           "AC".CTL_AV_OFFS_TD := "AM_PAR_INTERPOL" (x:=#act_x, phase:= #act_phase, interpol:= #act_interpol,
                           x_par:="PAR_X_VALUES_7".PAR, y_par:="PAR_CTL_OFFS_AVR_TD".PAR);

           "AC".CTL_AV_OFFS_T1 := "AM_PAR_INTERPOL" (x:=#act_x, phase:= #act_phase, interpol:= #act_interpol,
                           x_par:="PAR_X_VALUES_7".PAR, y_par:="PAR_CTL_OFFS_AVR_T1".PAR);
       END_IF;
END_FUNCTION

FUNCTION "AM_PAR_FNC_CAM" : Void   // FC234, SCL
{ S7_Optimized_Access := 'FALSE' }
VERSION : 0.0
// --------------------------------------------------------------------------------
//     program     :    AM_PAR_FNC_CAM
//     description :    Calculate all camera setpoints from function tables.
//     name        :    D.Bruess
//     date        :    21.10.99
// 
//     revision    :    1.00
//     name        :    D.Bruess
//     date        :    21.10.99
//                     (c) CGS
//     --------------------------------------------------------------------------------
   VAR_INPUT
      act_x : Real;   // actual x value, x > 0
      act_phase : Int;   // process phase, 0 ... 9
      act_interpol : Bool;   // TRUE = with interpolation
   END_VAR
   VAR_TEMP
      YAct : Real;
   END_VAR
BEGIN


       //refresh camera parameters from recipe tables in one second cycle
       //----------------------------------------------------------------
       IF "SysTick1s" THEN   
           "AC".SET_SEN_THR    := "AM_PAR_INTERPOL" (x:=#act_x, phase:= #act_phase, interpol:= #act_interpol,
                           x_par:="PAR_X_VALUES_10".PAR, y_par:="PAR_CAM_THR".PAR);

           "AC".SET_SEN_WDH    := "AM_PAR_INTERPOL" (x:=#act_x, phase:= #act_phase, interpol:= #act_interpol,
                        x_par:="PAR_X_VALUES_10".PAR, y_par:="PAR_CAM_WIN_SIZE_H".PAR);

           "AC".SET_SEN_HGT    := "AM_PAR_INTERPOL" (x:=#act_x, phase:= #act_phase, interpol:= #act_interpol,
                        x_par:="PAR_X_VALUES_10".PAR, y_par:="PAR_CAM_WIN_SIZE_V".PAR);

           "AC".SET_SEN_CTR_X  := "AM_PAR_INTERPOL" (x:=#act_x, phase:= #act_phase, interpol:= #act_interpol,
                        x_par:="PAR_X_VALUES_10".PAR, y_par:="PAR_CAM_WIN_POS_H".PAR);

           "AC".SET_SEN_CTR_Y  := "AM_PAR_INTERPOL" (x:=#act_x, phase:= #act_phase, interpol:= #act_interpol,
                        x_par:="PAR_X_VALUES_10".PAR, y_par:="PAR_CAM_WIN_POS_V".PAR);

           "AC".SET_SEN_OUT_RAD  := "AM_PAR_INTERPOL" (x:=#act_x, phase:= #act_phase, interpol:= #act_interpol,
                                                   x_par:="PAR_X_VALUES_10".PAR, y_par:="PAR_CAM_SET_OUT_RAD".PAR);

           "AC".SET_SEN_IN_RAD   := "AM_PAR_INTERPOL" (x:=#act_x, phase:= #act_phase, interpol:= #act_interpol,
                                                   x_par:="PAR_X_VALUES_10".PAR, y_par:="PAR_CAM_SET_IN_RAD".PAR);

           "AC".SET_SEN_SEQ_STR_AGL  := "AM_PAR_INTERPOL" (x:=#act_x, phase:= #act_phase, interpol:= #act_interpol,
                                                       x_par:="PAR_X_VALUES_10".PAR, y_par:="PAR_CAM_SET_SEQ_STR_AGL".PAR);

           "AC".SET_SEN_SEQ_STP_AGL  := "AM_PAR_INTERPOL" (x:=#act_x, phase:= #act_phase, interpol:= #act_interpol,
                                                       x_par:="PAR_X_VALUES_10".PAR, y_par:="PAR_CAM_SET_SEQ_STP_AGL".PAR);


           IF ((#act_phase ="APC".NECK) OR (#act_phase ="APC".SHOULDER) OR (#act_phase ="APC".BODY)) THEN

               "AC".XT_MENISCUS := "AM_PAR_INTERPOL"(x:=#act_x, phase:= #act_phase, interpol:= #act_interpol,
                                                   x_par:="PAR_X_VALUES_10".PAR, y_par:="PAR_XT_MEN".PAR);

           ELSE
               "AC".XT_MENISCUS := 0.0;
           END_IF;

           //stereo camera
           //-------------
           "AC".SET_ROI_CTR_X_SCAM   := "AM_PAR_INTERPOL" (x:=#act_x, phase:= #act_phase, interpol:= #act_interpol,
                        x_par:="PAR_X_VALUES_10".PAR, y_par:="PAR_SCAM_CTR_X_POS".PAR);

           "AC".SET_ROI_CTR_Y_SCAM   := "AM_PAR_INTERPOL" (x:=#act_x, phase:= #act_phase, interpol:= #act_interpol,
                        x_par:="PAR_X_VALUES_10".PAR, y_par:="PAR_SCAM_CTR_Y_POS".PAR);

           "AC".SET_CAM_2_THR    := "AM_PAR_INTERPOL" (x:=#act_x, phase:= #act_phase, interpol:= #act_interpol,
                           x_par:="PAR_X_VALUES_10".PAR, y_par:="PAR_CAM_2_THR".PAR);

       END_IF;
END_FUNCTION

FUNCTION "AM_PAR_FNC_AV_CR_ROT_CTL" : Void   // FC235, SCL
{ S7_Optimized_Access := 'FALSE' }
VERSION : 0.0
// --------------------------------------------------------------------------------
//     program     :    AM_PAR_FNC_AV_CR_ROT_CTL
//     description :    Calculate all pid parameter for average crucible rotation 
//                      control loop from function tables.
//     name        :    G. Eibelsh鋟ser
//     date        :    11.01.2001
// 
//     revision    :    
//     name        :    
//     date        :    
//                     (c) CGS
//     --------------------------------------------------------------------------------
   VAR_INPUT
      act_x : Real;   // actual x value, x > 0
      act_phase : Int;   // process phase, 0 ... 9
      act_interpol : Bool;   // TRUE = with interpolation
   END_VAR
   VAR_TEMP
      YAct : Real;
   END_VAR
BEGIN


      "AC".CTL_AV_CRUC_ROT_GN := "AM_PAR_INTERPOL" (x:=#act_x, phase:= #act_phase, interpol:= #act_interpol,
                            x_par:="PAR_X_VALUES_8".PAR, y_par:="PAR_CTRL_AV_CRUC_ROT_GN".PAR);

      "AC".CTL_AV_CRUC_ROT_TI := "AM_PAR_INTERPOL" (x:=#act_x, phase:= #act_phase, interpol:= #act_interpol,
                            x_par:="PAR_X_VALUES_8".PAR, y_par:="PAR_CTRL_AV_CRUC_ROT_TI".PAR);

      "AC".CTL_AV_CRUC_ROT_TD := "AM_PAR_INTERPOL" (x:=#act_x, phase:= #act_phase, interpol:= #act_interpol,
                            x_par:="PAR_X_VALUES_8".PAR, y_par:="PAR_CTRL_AV_CRUC_ROT_TD".PAR);

      "AC".CTL_AV_CRUC_ROT_T1 := "AM_PAR_INTERPOL" (x:=#act_x, phase:= #act_phase, interpol:= #act_interpol,
                            x_par:="PAR_X_VALUES_8".PAR, y_par:="PAR_CTRL_AV_CRUC_ROT_T1".PAR);
END_FUNCTION

FUNCTION "AM_PAR_FNC_PD" : Void   // FC240, SCL
{ S7_Optimized_Access := 'FALSE' }
VERSION : 0.0
// --------------------------------------------------------------------------------
//     program     :    AM_PAR_FNC_PD
//     description :    Calculate all from function tables for PUMP DOWN process.
//     name        :    D.Bruess
//     date        :    21.10.99
// 
//     revision    :    1.00
//     name        :    D.Bruess
//     date        :    21.10.99
//                     (c) CGS
//     --------------------------------------------------------------------------------
   VAR_INPUT
      act_x_value : Real;   // actual x value, x > 0
   END_VAR
   VAR_TEMP
      YAct : Real;
      act_phase_number : Int;
   END_VAR
BEGIN


     #act_phase_number := "APC".PUMP_DOWN;

     // main page
     // ---------
     "AM_SET_V2" (act_phase := #act_phase_number);
     "AC".XT_MENISCUS := 0.0;

     // page 1
     // ------

     // page 2
     // ------

     // page 3
     // ------

     // page 4
     // ------

     // page 5
     // ------

     // page 6
     // ------

     // page 7
     // ------

     // page 8
     // ------

     // page 9
     // ------

     // page 10
     // ------
END_FUNCTION

FUNCTION "AM_PAR_FNC_ME" : Void   // FC241, SCL
{ S7_Optimized_Access := 'FALSE' }
VERSION : 0.0
// --------------------------------------------------------------------------------
//     program     :    AM_PAR_FNC_ME
//     description :    Calculate all from function tables for MELTING process.
//     name        :    D.Bruess
//     date        :    21.10.99
// 
//     revision    :    1.00
//     name        :    D.Bruess
//     date        :    21.10.99
//                     (c) CGS
//     --------------------------------------------------------------------------------
   VAR_INPUT
      act_x_value : Real;   // actual x value, x > 0
   END_VAR
   VAR_TEMP
      YAct : Real;
      act_phase_number : Int;
   END_VAR
BEGIN


     #act_phase_number := "APC".MELTING;

     // main page
     // ---------
     "AM_SET_V2" (act_phase := #act_phase_number);

     // page 1
     // ------
   (*YAct := AM_PAR_INTERPOL 
               (x:=act_x_value, phase:= act_phase_number, interpol:= FALSE,
                      x_par:=PAR_X_VALUES_1.PAR, y_par:=PAR_TIME.PAR);   *)

     "AV".SET_CR_POS := "AM_PAR_INTERPOL" 
               (x:=#act_x_value, phase:= #act_phase_number, interpol:= FALSE,
                      x_par:="PAR_X_VALUES_1".PAR, y_par:="PAR_CR_POS".PAR);

     "AV".SET_CR_SPD := "AM_PAR_INTERPOL" 
               (x:=#act_x_value, phase:= #act_phase_number, interpol:= FALSE,
                      x_par:="PAR_X_VALUES_1".PAR, y_par:="PAR_CR_SPD".PAR);

     "AC".SET_HTR_1_PWR := "AM_PAR_INTERPOL" 
               (x:=#act_x_value, phase:= #act_phase_number, interpol:= FALSE,
                      x_par:="PAR_X_VALUES_1".PAR, y_par:="PAR_HTR_1_PWR".PAR);

     "AC".SET_HTR_2_PWR := "AM_PAR_INTERPOL" 
               (x:=#act_x_value, phase:= #act_phase_number, interpol:= FALSE,
                      x_par:="PAR_X_VALUES_1".PAR, y_par:="PAR_HTR_2_PWR".PAR);

     "AC".SET_MOB_FDR_VIB_FRQ := "AM_PAR_INTERPOL" 
               (x:=#act_x_value, phase:= #act_phase_number, interpol:= FALSE,
                      x_par:="PAR_X_VALUES_1".PAR, y_par:="PAR_FDR_VIB_FRQ".PAR);





     // page 2
     // ------  

     // page 3
     // ------  
     "AM_PAR_FNC_ROT"
               (act_x:=#act_x_value, act_phase:=#act_phase_number, act_interpol:=FALSE);

     // page 4
     // ------
     "AM_PAR_FNC_GAS"
               (act_x:=#act_x_value, act_phase:=#act_phase_number, act_interpol:=FALSE);

     // page 5
     // ------
     "AM_PAR_FNC_MAG"
               (act_x:=#act_x_value, act_phase:=#act_phase_number, act_interpol:=FALSE);

     // page 6
     // ------

     // page 7
     // ------

     // page 8
     // ------

     // page 9
     // ------

     // page 10
     // ------
     "AM_PAR_FNC_CAM"
               (act_x:=#act_x_value, act_phase:=#act_phase_number, act_interpol:=FALSE);
END_FUNCTION

FUNCTION "AM_PAR_FNC_DI" : Void   // FC242, SCL
{ S7_Optimized_Access := 'FALSE' }
VERSION : 0.0
// --------------------------------------------------------------------------------
//     program     :    AM_PAR_FNC_DI
//     description :    Calculate all from function tables for DIPPING process.
//     name        :    D.Bruess
//     date        :    22.10.99
// 
//     revision    :    1.00
//     name        :    D.Bruess
//     date        :    22.10.99
//                     (c) CGS
//     --------------------------------------------------------------------------------
   VAR_INPUT
      act_x_value : Real;   // actual x value, x > 0
   END_VAR
   VAR_TEMP
      YAct : Real;
      act_phase_number : Int;
   END_VAR
BEGIN


     #act_phase_number := "APC".DIPPING;

     // main page
     // ---------
     "AM_SET_V2" (act_phase := #act_phase_number);

     // page 1
     // ------
   (*YAct := AM_PAR_INTERPOL (x:=act_x_value, phase:= act_phase_number, interpol:= FALSE,
                      x_par:=PAR_X_VALUES_1.PAR, y_par:=PAR_TIME.PAR);   *)

     // page 2
     // ------                 

     // page 3
     // ------  
     "AM_PAR_FNC_ROT"
               (act_x:=#act_x_value, act_phase:=#act_phase_number, act_interpol:=FALSE);

     // page 4
     // ------
     "AM_PAR_FNC_GAS" 
               (act_x:=#act_x_value, act_phase:=#act_phase_number, act_interpol:=FALSE);

     // page 5
     // ------
     "AM_PAR_FNC_MAG"
               (act_x:=#act_x_value, act_phase:=#act_phase_number, act_interpol:=FALSE);

     // page 6
     // ------

     // page 7
     // ------
     "AC".CTL_MLT_TMP_1_GN := "AM_PAR_INTERPOL" 
               (x:=#act_x_value, phase:= #act_phase_number, interpol:= FALSE,
                      x_par:="PAR_X_VALUES_7".PAR, y_par:="PAR_CTRL_MLT_TMP_1_GN".PAR);

     "AC".CTL_MLT_TMP_1_TI := "AM_PAR_INTERPOL" 
               (x:=#act_x_value, phase:= #act_phase_number, interpol:= FALSE,
                      x_par:="PAR_X_VALUES_7".PAR, y_par:="PAR_CTRL_MLT_TMP_1_TI".PAR);

     "AC".CTL_MLT_TMP_1_TD := "AM_PAR_INTERPOL"
               (x:=#act_x_value, phase:= #act_phase_number, interpol:= FALSE,
                      x_par:="PAR_X_VALUES_7".PAR, y_par:="PAR_CTRL_MLT_TMP_1_TD".PAR);

     "AC".CTL_MLT_TMP_1_T1 := "AM_PAR_INTERPOL"
               (x:=#act_x_value, phase:= #act_phase_number, interpol:= FALSE,
                      x_par:="PAR_X_VALUES_7".PAR, y_par:="PAR_CTRL_MLT_TMP_1_T1".PAR);

     // page 8
     // ------                 

     // page 9
     // ------
     "AC".PWR_COEFF_2 := "AM_PAR_INTERPOL" 
               (x:=#act_x_value, phase:= #act_phase_number, interpol:= FALSE,
                      x_par:="PAR_X_VALUES_9".PAR, y_par:="PAR_PWR_COEFF_2".PAR);

     // page 10
     // ------
     "AM_PAR_FNC_CAM" 
               (act_x:=#act_x_value, act_phase:=#act_phase_number, act_interpol:=FALSE);
END_FUNCTION

FUNCTION "AM_PAR_FNC_NE" : Void   // FC243, SCL
{ S7_Optimized_Access := 'FALSE' }
VERSION : 0.0
// --------------------------------------------------------------------------------
//     program     :    AM_PAR_FNC_NE
//     description :    Calculate all from function tables for NECK process.
//     name        :    D.Bruess
//     date        :    22.10.99
// 
//     revision    :    1.00
//     name        :    D.Bruess
//     date        :    22.10.99
//                     (c) CGS
//     --------------------------------------------------------------------------------
   VAR_INPUT
      act_x_value : Real;   // actual x value, x > 0
   END_VAR
   VAR_TEMP
      YAct : Real;
      act_phase_number : Int;
   END_VAR
BEGIN


     #act_phase_number := "APC".NECK;

     // main page
     // ---------
     "AM_SET_V2" (act_phase := #act_phase_number);

     // page 1
     // ------
     "AC".SET_AVG_SPD := "AM_PAR_INTERPOL" 
               (x:=#act_x_value, phase:= #act_phase_number, interpol:= TRUE,
                      x_par:="PAR_X_VALUES_1".PAR, y_par:="PAR_AV_SPD".PAR);

     "AC".SET_XT_SPD_DEV_1 := "AM_PAR_INTERPOL" 
               (x:=#act_x_value, phase:= #act_phase_number, interpol:= TRUE,
                      x_par:="PAR_X_VALUES_1".PAR, y_par:="PAR_AV_SPD_DEV_1".PAR);

     "AC".SET_XT_SPD_DEV_2 := "AM_PAR_INTERPOL" 
               (x:=#act_x_value, phase:= #act_phase_number, interpol:= TRUE,
                      x_par:="PAR_X_VALUES_1".PAR, y_par:="PAR_AV_SPD_DEV_2".PAR);

     "AV".SET_HTR_1_TMP_INC := "AM_PAR_INTERPOL" 
               (x:=#act_x_value, phase:= #act_phase_number, interpol:= TRUE,
                      x_par:="PAR_X_VALUES_1".PAR, y_par:="PAR_HTR_1_TMP".PAR);

     "AV".SET_HTR_2_PWR_INC := "AM_PAR_INTERPOL" 
               (x:=#act_x_value, phase:= #act_phase_number, interpol:= TRUE,
                      x_par:="PAR_X_VALUES_1".PAR, y_par:="PAR_HTR_2_PWR".PAR);

     // page 2
     // ------
     "AV".SET_XT_DIA := "AM_PAR_INTERPOL" 
               (x:=#act_x_value, phase:= #act_phase_number, interpol:= TRUE,
                      x_par:="PAR_X_VALUES_2".PAR, y_par:="PAR_XT_DIA".PAR);

     // page 3
     // ------  
     "AM_PAR_FNC_ROT"
               (act_x:=#act_x_value, act_phase:=#act_phase_number, act_interpol:=TRUE);

     // page 4
     // ------
     "AM_PAR_FNC_GAS" 
               (act_x:=#act_x_value, act_phase:=#act_phase_number, act_interpol:=TRUE);

     // page 5
     // ------
     "AM_PAR_FNC_MAG"
               (act_x:=#act_x_value, act_phase:=#act_phase_number, act_interpol:=TRUE);

     // page 6
     // ------

     // page 7
     // ------
     "AM_PAR_FNC_CTL" 
               (act_x:=#act_x_value, act_phase:=#act_phase_number, act_interpol:=TRUE);

     // page 8
     // ------          

     // page 9
     // ------
     "AC".PWR_COEFF_2 := "AM_PAR_INTERPOL" 
               (x:=#act_x_value, phase:= #act_phase_number, interpol:= TRUE,
                      x_par:="PAR_X_VALUES_9".PAR, y_par:="PAR_PWR_COEFF_2".PAR);

     // page 10
     // ------
     "AM_PAR_FNC_CAM" 
               (act_x:=#act_x_value, act_phase:=#act_phase_number, act_interpol:= TRUE);
END_FUNCTION

FUNCTION "AM_PAR_FNC_SH" : Void   // FC244, SCL
{ S7_Optimized_Access := 'FALSE' }
VERSION : 0.0
// --------------------------------------------------------------------------------
//     program     :    AM_PAR_FNC_SH
//     description :    Calculate all from function tables for SHOULDER process.
//     name        :    D.Bruess
//     date        :    22.10.99
// 
//     revision    :    1.00
//     name        :    D.Bruess
//     date        :    22.10.99
//                     (c) CGS
//     --------------------------------------------------------------------------------
   VAR_INPUT
      act_x_value : Real;   // actual x value, x > 0
   END_VAR
   VAR_TEMP
      YAct : Real;
      act_phase_number : Int;
   END_VAR
BEGIN


     #act_phase_number := "APC".SHOULDER;

     // main page
     // ---------
     "AM_SET_V2" (act_phase := #act_phase_number);

     // page 1
     // ------
     "AC".SET_GRW_RTE := "AM_PAR_INTERPOL" 
               (x:=#act_x_value, phase:= #act_phase_number, interpol:= TRUE,
                      x_par:="PAR_X_VALUES_1".PAR, y_par:="PAR_XT_GRO".PAR);


     IF "DV".TRANS_SH_BY_FLAG AND "CNF".CONF_SH_PAR_FNCT THEN   //transition to body? SH-Par as function of length? 
       "AC".SET_XT_SPD := "PAR_MAIN".SH_BODY_TRANS_SPD;        
     ELSE                                                  
       "AC".SET_XT_SPD := "AM_PAR_INTERPOL" 
                (x:=#act_x_value, phase:= #act_phase_number, interpol:= TRUE,
                       x_par:="PAR_X_VALUES_1".PAR, y_par:="PAR_XT_SPD".PAR);
     END_IF;                    

     "AC".SET_AVG_CRUC_ROT := "AM_PAR_INTERPOL" 
               (x:=#act_x_value, phase:= #act_phase_number, interpol:= TRUE,
                      x_par:="PAR_X_VALUES_1".PAR, y_par:="PAR_AV_CRUC_ROT".PAR);

     "AC".SET_CRUC_ROT_DEV_1 := "AM_PAR_INTERPOL" 
               (x:=#act_x_value, phase:= #act_phase_number, interpol:= TRUE,
                      x_par:="PAR_X_VALUES_1".PAR, y_par:="PAR_AV_CRUC_ROT_DEV_1".PAR);

     "AC".SET_CRUC_ROT_DEV_2 := "AM_PAR_INTERPOL" 
               (x:=#act_x_value, phase:= #act_phase_number, interpol:= TRUE,
                      x_par:="PAR_X_VALUES_1".PAR, y_par:="PAR_AV_CRUC_ROT_DEV_2".PAR);

     "AV".SET_HTR_1_TMP_INC := "AM_PAR_INTERPOL" 
               (x:=#act_x_value, phase:= #act_phase_number, interpol:= TRUE,
                      x_par:="PAR_X_VALUES_1".PAR, y_par:="PAR_HTR_1_TMP".PAR);

     "AV".SET_HTR_2_PWR_INC := "AM_PAR_INTERPOL" 
               (x:=#act_x_value, phase:= #act_phase_number, interpol:= TRUE,
                      x_par:="PAR_X_VALUES_1".PAR, y_par:="PAR_HTR_2_PWR".PAR);

     // page 2
     // ------  

     // page 3
     // ------  
     "AM_PAR_FNC_ROT"
               (act_x:=#act_x_value, act_phase:=#act_phase_number, act_interpol:=TRUE);

     // page 4
     // ------
     "AM_PAR_FNC_GAS" 
               (act_x:=#act_x_value, act_phase:=#act_phase_number, act_interpol:=TRUE);

     // page 5
     // ------
     "AM_PAR_FNC_MAG"
               (act_x:=#act_x_value, act_phase:=#act_phase_number, act_interpol:=TRUE);

     // page 6
     // ------
     "AC".SET_CR_SPD_COF := "AM_PAR_INTERPOL" 
               (x:=#act_x_value, phase:= #act_phase_number, interpol:= TRUE,
                      x_par:="PAR_X_VALUES_6".PAR, y_par:="PAR_CRSPD_COEFF".PAR);


     "AC".CTL_MLT_LVL_GN := "AM_PAR_INTERPOL" 
               (x:=#act_x_value, phase:= #act_phase_number, interpol:= TRUE,
                      x_par:="PAR_X_VALUES_6".PAR, y_par:="PAR_CTRL_MLT_LVL_GN".PAR);


     "AC".SET_MLT_LVL_INC := "AM_PAR_INTERPOL" 
               (x:=#act_x_value, phase:= #act_phase_number, interpol:= TRUE,
                      x_par:="PAR_X_VALUES_6".PAR, y_par:="PAR_MLT_LVL_INC".PAR);





     // page 7
     // ------
     "AC".CTL_GRO_GN := "AM_PAR_INTERPOL" 
               (x:=#act_x_value, phase:= #act_phase_number, interpol:= TRUE,
                      x_par:="PAR_X_VALUES_7".PAR, y_par:="PAR_CTRL_GRO_GN".PAR);

     "AC".CTL_GRO_TI := "AM_PAR_INTERPOL" 
               (x:=#act_x_value, phase:= #act_phase_number, interpol:= TRUE,
                      x_par:="PAR_X_VALUES_7".PAR, y_par:="PAR_CTRL_GRO_TI".PAR);

     "AC".CTL_GRO_TD := "AM_PAR_INTERPOL" 
               (x:=#act_x_value, phase:= #act_phase_number, interpol:= TRUE,
                      x_par:="PAR_X_VALUES_7".PAR, y_par:="PAR_CTRL_GRO_TD".PAR);

     "AC".CTL_GRO_T1 := "AM_PAR_INTERPOL" 
               (x:=#act_x_value, phase:= #act_phase_number, interpol:= TRUE,
                      x_par:="PAR_X_VALUES_7".PAR, y_par:="PAR_CTRL_GRO_T1".PAR);

     // page 8
     // ------
     "AM_PAR_FNC_AV_CR_ROT_CTL" 
               (act_x:=#act_x_value, act_phase:=#act_phase_number, act_interpol:=TRUE);

     // page 9
     // ------
     "AC".PWR_COEFF_2 := "AM_PAR_INTERPOL" 
               (x:=#act_x_value, phase:= #act_phase_number, interpol:= TRUE,
                      x_par:="PAR_X_VALUES_9".PAR, y_par:="PAR_PWR_COEFF_2".PAR);

     // page 10
     // -------
     "AM_PAR_FNC_CAM" 
               (act_x:=#act_x_value, act_phase:=#act_phase_number, act_interpol:= TRUE);
END_FUNCTION

FUNCTION "AM_PAR_FNC_BY" : Void   // FC245, SCL
{ S7_Optimized_Access := 'FALSE' }
VERSION : 0.0
// --------------------------------------------------------------------------------
//     program     :    AM_PAR_FNC_BY
//     description :    Calculate all from function tables for BODY process.
//     name        :    D.Bruess
//     date        :    22.10.99
// 
//     revision    :    1.00
//     name        :    D.Bruess
//     date        :    22.10.99
//                     (c) CGS
//     --------------------------------------------------------------------------------
   VAR_INPUT
      act_x_value : Real;   // actual x value, x > 0
   END_VAR
   VAR_TEMP
      YAct : Real;
      act_phase_number : Int;
   END_VAR
BEGIN


     #act_phase_number := "APC".BODY;

     // main page
     // ---------
     "AM_SET_V2" (act_phase := #act_phase_number);

     // page 1
     // ------
     "AC".SET_AVG_SPD := "AM_PAR_INTERPOL" 
               (x:=#act_x_value, phase:= #act_phase_number, interpol:= TRUE,
                      x_par:="PAR_X_VALUES_1".PAR, y_par:="PAR_AV_SPD".PAR);

     "AC".SET_XT_SPD_DEV_1 := "AM_PAR_INTERPOL" 
               (x:=#act_x_value, phase:= #act_phase_number, interpol:= TRUE,
                      x_par:="PAR_X_VALUES_1".PAR, y_par:="PAR_AV_SPD_DEV_1".PAR);

     "AC".SET_XT_SPD_DEV_2 := "AM_PAR_INTERPOL" 
               (x:=#act_x_value, phase:= #act_phase_number, interpol:= TRUE,
                      x_par:="PAR_X_VALUES_1".PAR, y_par:="PAR_AV_SPD_DEV_2".PAR);

     "AC".SET_AVG_CRUC_ROT := "AM_PAR_INTERPOL" 
               (x:=#act_x_value, phase:= #act_phase_number, interpol:= TRUE,
                      x_par:="PAR_X_VALUES_1".PAR, y_par:="PAR_AV_CRUC_ROT".PAR);

     "AC".SET_CRUC_ROT_DEV_1 := "AM_PAR_INTERPOL" 
               (x:=#act_x_value, phase:= #act_phase_number, interpol:= TRUE,
                      x_par:="PAR_X_VALUES_1".PAR, y_par:="PAR_AV_CRUC_ROT_DEV_1".PAR);

     "AC".SET_CRUC_ROT_DEV_2 := "AM_PAR_INTERPOL" 
               (x:=#act_x_value, phase:= #act_phase_number, interpol:= TRUE,
                      x_par:="PAR_X_VALUES_1".PAR, y_par:="PAR_AV_CRUC_ROT_DEV_2".PAR);

     "AV".SET_HTR_1_TMP_INC := "AM_PAR_INTERPOL" 
               (x:=#act_x_value, phase:= #act_phase_number, interpol:= TRUE,
                      x_par:="PAR_X_VALUES_1".PAR, y_par:="PAR_HTR_1_TMP".PAR);

     "AV".SET_HTR_2_PWR_INC := "AM_PAR_INTERPOL" 
               (x:=#act_x_value, phase:= #act_phase_number, interpol:= TRUE,
                      x_par:="PAR_X_VALUES_1".PAR, y_par:="PAR_HTR_2_PWR".PAR);

     // page 2
     // ------
     "AV".SET_XT_DIA := "AM_PAR_INTERPOL" 
               (x:=#act_x_value, phase:= #act_phase_number, interpol:= TRUE,
                      x_par:="PAR_X_VALUES_2".PAR, y_par:="PAR_XT_DIA".PAR);

     // page 3
     // ------  
     "AM_PAR_FNC_ROT"
               (act_x:=#act_x_value, act_phase:=#act_phase_number, act_interpol:=TRUE);

     // page 4
     // ------
     "AM_PAR_FNC_GAS" 
               (act_x:=#act_x_value, act_phase:=#act_phase_number, act_interpol:=TRUE);

     // page 5
     // ------
     "AM_PAR_FNC_MAG"
               (act_x:=#act_x_value, act_phase:=#act_phase_number, act_interpol:=TRUE);

     // page 6
     // ------
     "AC".SET_CR_SPD_COF := "AM_PAR_INTERPOL" 
               (x:=#act_x_value, phase:= #act_phase_number, interpol:= TRUE,
                      x_par:="PAR_X_VALUES_6".PAR, y_par:="PAR_CRSPD_COEFF".PAR);


     "AC".CTL_MLT_LVL_GN := "AM_PAR_INTERPOL" 
               (x:=#act_x_value, phase:= #act_phase_number, interpol:= TRUE,
                      x_par:="PAR_X_VALUES_6".PAR, y_par:="PAR_CTRL_MLT_LVL_GN".PAR);


     "AC".SET_MLT_LVL_INC := "AM_PAR_INTERPOL" 
               (x:=#act_x_value, phase:= #act_phase_number, interpol:= TRUE,
                      x_par:="PAR_X_VALUES_6".PAR, y_par:="PAR_MLT_LVL_INC".PAR);


     // page 7
     // ------
     "AM_PAR_FNC_CTL" 
               (act_x:=#act_x_value, act_phase:=#act_phase_number, act_interpol:=TRUE);

     // page 8
     // ------
     "AM_PAR_FNC_AV_CR_ROT_CTL" 
               (act_x:=#act_x_value, act_phase:=#act_phase_number, act_interpol:=TRUE);

     // page 9
     // ------
     "AC".PWR_COEFF_2 := "AM_PAR_INTERPOL" 
               (x:=#act_x_value, phase:= #act_phase_number, interpol:= TRUE,
                      x_par:="PAR_X_VALUES_9".PAR, y_par:="PAR_PWR_COEFF_2".PAR);

     // page 10
     // -------
     "AM_PAR_FNC_CAM" 
               (act_x:=#act_x_value, act_phase:=#act_phase_number, act_interpol:= TRUE);

       // page 11
       // -------
       "AC".CTL_DIA_TMP_GN :=    "AM_PAR_INTERPOL"(x           := #act_x_value, 
                                               phase       := #act_phase_number, 
                                               interpol    := TRUE,
                                               x_par       := "PAR_X_VALUES_11".PAR, 
                                               y_par       := "PAR_CTRL_DIA_TMP_GN".PAR);

       "AC".CTL_DIA_TMP_TI :=    "AM_PAR_INTERPOL"(x           := #act_x_value, 
                                               phase       := #act_phase_number, 
                                               interpol    := TRUE,
                                               x_par       := "PAR_X_VALUES_11".PAR, 
                                               y_par       := "PAR_CTRL_DIA_TMP_TI".PAR);

       "AC".CTL_DIA_TMP_TD :=    "AM_PAR_INTERPOL"(x           := #act_x_value, 
                                               phase       := #act_phase_number, 
                                               interpol    := TRUE,
                                               x_par       := "PAR_X_VALUES_11".PAR, 
                                               y_par       := "PAR_CTRL_DIA_TMP_TD".PAR);

       "AC".CTL_DIA_TMP_T1 :=    "AM_PAR_INTERPOL"(x           := #act_x_value, 
                                               phase       := #act_phase_number, 
                                               interpol    := TRUE,
                                               x_par       := "PAR_X_VALUES_11".PAR, 
                                               y_par       := "PAR_CTRL_DIA_TMP_T1".PAR);
END_FUNCTION

FUNCTION "AM_PAR_FNC_EC" : Void   // FC246, SCL
{ S7_Optimized_Access := 'FALSE' }
VERSION : 0.0
// --------------------------------------------------------------------------------
//     program     :    AM_PAR_FNC_EC
//     description :    Calculate all from function tables for ENDCONE process.
//     name        :    D.Bruess
//     date        :    22.10.99
// 
//     revision    :    1.00
//     name        :    D.Bruess
//     date        :    22.10.99
//                     (c) CGS
//     --------------------------------------------------------------------------------
   VAR_INPUT
      act_x_value : Real;   // actual x value, x > 0
   END_VAR
   VAR_TEMP
      YAct : Real;
      act_phase_number : Int;
   END_VAR
BEGIN


     #act_phase_number := "APC".ENDCONE;

     // main page
     // ---------
     "AM_SET_V2" (act_phase := #act_phase_number);

     // page 1
     // ------
     "AV".SET_XT_SPD := "AM_PAR_INTERPOL" 
               (x:=#act_x_value, phase:= #act_phase_number, interpol:= TRUE,
                      x_par:="PAR_X_VALUES_1".PAR, y_par:="PAR_XT_SPD".PAR);

     "AV".SET_CR_SPD := "AM_PAR_INTERPOL" 
               (x:=#act_x_value, phase:= #act_phase_number, interpol:= TRUE,
                      x_par:="PAR_X_VALUES_1".PAR, y_par:="PAR_CR_SPD".PAR);

     "AV".SET_HTR_1_TMP_INC := "AM_PAR_INTERPOL" 
               (x:=#act_x_value, phase:= #act_phase_number, interpol:= TRUE,
                      x_par:="PAR_X_VALUES_1".PAR, y_par:="PAR_HTR_1_TMP".PAR);

     "AV".SET_HTR_2_PWR_INC := "AM_PAR_INTERPOL" 
               (x:=#act_x_value, phase:= #act_phase_number, interpol:= TRUE,
                      x_par:="PAR_X_VALUES_1".PAR, y_par:="PAR_HTR_2_PWR".PAR);

     // page 2
     // ------  

     // page 3
     // ------
     "AM_PAR_FNC_ROT"
               (act_x:=#act_x_value, act_phase:=#act_phase_number, act_interpol:=TRUE);

     // page 4
     // ------
     "AM_PAR_FNC_GAS" 
               (act_x:=#act_x_value, act_phase:=#act_phase_number, act_interpol:=TRUE);

     // page 5
     // ------
     "AM_PAR_FNC_MAG"
               (act_x:=#act_x_value, act_phase:=#act_phase_number, act_interpol:=TRUE);

     // page 6
     // ------

     // page 7
     // ------

     // page 8
     // ------

     // page 9
     // ------
     "AC".PWR_COEFF_2 := "AM_PAR_INTERPOL" 
               (x:=#act_x_value, phase:= #act_phase_number, interpol:= TRUE,
                      x_par:="PAR_X_VALUES_9".PAR, y_par:="PAR_PWR_COEFF_2".PAR);

     // page 10
     // -------

     "AC".XT_MENISCUS := 0.0;
END_FUNCTION

FUNCTION "AM_PAR_FNC_SD" : Void   // FC247, SCL
{ S7_Optimized_Access := 'FALSE' }
VERSION : 0.0
// --------------------------------------------------------------------------------
//     program     :    AM_PAR_FNC_SD
//     description :    Calculate all from function tables for SHUT DOWN process.
//     name        :    D.Bruess
//     date        :    22.10.99
// 
//     revision    :    1.00
//     name        :    D.Bruess
//     date        :    22.10.99
//                     (c) CGS
//     --------------------------------------------------------------------------------
   VAR_INPUT
      act_x_value : Real;   // actual x value, x > 0
   END_VAR
   VAR_TEMP
      YAct : Real;
      act_phase_number : Int;
   END_VAR
BEGIN


     #act_phase_number := "APC".SHUT_DOWN;

     // main page
     // ---------
     "AM_SET_V2" (act_phase := #act_phase_number);

     // page 1
     // ------
   (*YAct := AM_PAR_INTERPOL 
               (x:=act_x_value, phase:= act_phase_number, interpol:= FALSE,
                      x_par:=PAR_X_VALUES_1.PAR, y_par:=PAR_TIME.PAR);   *)

     "AV".SET_XT_POS := "AM_PAR_INTERPOL" 
               (x:=#act_x_value, phase:= #act_phase_number, interpol:= FALSE,
                      x_par:="PAR_X_VALUES_1".PAR, y_par:="PAR_XT_POS".PAR);

     "AV".SET_XT_SPD := "AM_PAR_INTERPOL" 
               (x:=#act_x_value, phase:= #act_phase_number, interpol:= FALSE,
                      x_par:="PAR_X_VALUES_1".PAR, y_par:="PAR_XT_SPD".PAR);

     "AV".SET_CR_POS := "AM_PAR_INTERPOL" 
               (x:=#act_x_value, phase:= #act_phase_number, interpol:= FALSE,
                      x_par:="PAR_X_VALUES_1".PAR, y_par:="PAR_CR_POS".PAR);

     "AV".SET_CR_SPD := "AM_PAR_INTERPOL" 
               (x:=#act_x_value, phase:= #act_phase_number, interpol:= FALSE,
                      x_par:="PAR_X_VALUES_1".PAR, y_par:="PAR_CR_SPD".PAR);

     "AC".SET_HTR_1_PWR := "AM_PAR_INTERPOL" 
               (x:=#act_x_value, phase:= #act_phase_number, interpol:= FALSE,
                      x_par:="PAR_X_VALUES_1".PAR, y_par:="PAR_HTR_1_PWR".PAR);

     // page 2
     // ------  

     // page 3
     // ------
     "AM_PAR_FNC_ROT"
               (act_x:=#act_x_value, act_phase:=#act_phase_number, act_interpol:=FALSE);


     // page 4 (AV.xxx used for AM_PRS_CTRL() )
     // ------
     "AV".SET_GAS_1_FLW := "AM_PAR_INTERPOL"
               (x:=#act_x_value, phase:= #act_phase_number, interpol:= FALSE,
                      x_par:="PAR_X_VALUES_4".PAR, y_par:="PAR_GAS_1_FLW".PAR);

     "AV".SET_GAS_2_FLW := "AM_PAR_INTERPOL"
               (x:=#act_x_value, phase:= #act_phase_number, interpol:= FALSE,
                      x_par:="PAR_X_VALUES_4".PAR, y_par:="PAR_GAS_2_FLW".PAR);

     "AV".SET_PRS_FCH := "AM_PAR_INTERPOL"
               (x:=#act_x_value, phase:= #act_phase_number, interpol:= FALSE,
                      x_par:="PAR_X_VALUES_4".PAR, y_par:="PAR_PRS".PAR);

     // page 5
     // ------
     "AM_PAR_FNC_MAG"
               (act_x:=#act_x_value, act_phase:=#act_phase_number, act_interpol:=FALSE);

     // page 6
     // ------

     // page 7
     // ------

     // page 8
     // ------

     // page 9
     // ------
     "AC".PWR_COEFF_2 := "AM_PAR_INTERPOL" 
               (x:=#act_x_value, phase:= #act_phase_number, interpol:= FALSE,
                      x_par:="PAR_X_VALUES_9".PAR, y_par:="PAR_PWR_COEFF_2".PAR);

     // page 10
     // -------

     "AC".XT_MENISCUS := 0.0;
END_FUNCTION

FUNCTION "AM_PAR_FNC_RE" : Void   // FC248, SCL
{ S7_Optimized_Access := 'FALSE' }
VERSION : 0.0
// --------------------------------------------------------------------------------
//     program     :    AM_PAR_FNC_RE
//     description :    Calculate all from function tables for REMOVAL process.
//     name        :    G. Eibelsh鋟ser
//     date        :    31.07.2012
// 
//                     (c) PVA TePla AG
//     --------------------------------------------------------------------------------
   VAR_TEMP
      YAct : Real;
      act_phase_number : Int;
   END_VAR
BEGIN


     #act_phase_number := "APC".REMOVAL;

     // main page
     // ---------

     "AM_SET_V2" (act_phase := #act_phase_number);

     "AC".SET_GAS_1_FLW     := "PAR_MAIN".RC_GAS_1_FLW;
     "AC".SET_GAS_2_FLW     := "PAR_MAIN".RC_GAS_2_FLW;
     "AC".SET_CLF_PRS       := "PAR_MAIN".RC_PRS;

     "AV".SET_MAG_1_CUR     := "PAR_MAIN".RC_MAG_AV_CUR;
     "AV".SET_MAG_RATIO_CUR := "PAR_MAIN".RC_MAG_RATIO_CUR;
END_FUNCTION

FUNCTION "AM_PAR_INTERPOL" : Real   // FC254, SCL
{ S7_Optimized_Access := 'FALSE' }
VERSION : 0.0
// --------------------------------------------------------------------------------
//     program     :    AM_INTERPOLATION
//     description :    Calculate y value from x/y function table.
//     name        :    D.Bruess
//     date        :    18.10.99
// 
//     revision    :    process phase 1 ...10
//     name        :    D.Bruess
//     date        :    12.11.99
//                     (c) CGS
//     --------------------------------------------------------------------------------
   VAR_INPUT
      x : Real;   // actual x value, x > 0
      phase : Int;   // process phase, 1 ... 10
      interpol : Bool;   // TRUE = with interpolation
      x_par : Array[1..10, 1..21] of Real;   // array with x values
      y_par : Array[1..10, 1..21] of Real;   // array with y values
   END_VAR
   VAR_TEMP
      x1 : Real;
      x2 : Real;
      y1 : Real;
      y2 : Real;
      y : Real;
      i : Int;
      found : Int;
   END_VAR
BEGIN

     IF ((#phase > 10) OR (#phase < 1)) THEN       // invalid phase number ?
       #y := 0.0;
     ELSE;

       IF (#x < 0.0) THEN                        // invalid x value ?
         #y := #y_par[#phase,1];
       ELSE

         // search for interval
         #i := 1;
         #found := 0;

         WHILE #found = 0 DO

           #x1 := #x_par[#phase,#i];
           #x2 := #x_par[#phase,#i+1];
           #y1 := #y_par[#phase,#i];
           #y2 := #y_par[#phase,#i+1];

           IF (#x <= #x1) THEN                    // below x1 ?

             #y := #y1;  
             #found := 1;
           ELSE
             IF (#x < #x2) THEN                    // x1<x<x2 ?
               IF (#interpol = TRUE) THEN
                 #y := #y1 + ((#y2-#y1)/(#x2-#x1))*(#x-#x1);
               ELSE
                 #y := #y1;
               END_IF;
               #found := 1;

             ELSE                                 // x>=x2                           

               IF (#x2=0.0) THEN                   // last x[i] because next x=0 ?
                 #y := #y1;
                 #found := 1;
               ELSE
                 IF (#i = 20) THEN                 // last x[i] because i = 20 ?
                   #y := #y2;
                   #found := 1;

                 ELSE
                   #i := #i + 1;                    // next x[i]
                   #found := 0;

                 END_IF;

               END_IF;
              END_IF;
             END_IF;
           END_WHILE;
         END_IF;
       END_IF;


     #AM_PAR_INTERPOL := #y;
END_FUNCTION

FUNCTION "SM_RESTART_CALL" : Void   // FC256, SCL
{ S7_Optimized_Access := 'FALSE' }
VERSION : 0.0
// --------------------------------------------------------------------------------
//     program     :    SM_RESTART_CALL
//     description :    call functions for restart       
//     name        :    K. Kalkowski
//     date        :    04.11.98
// 
//     revision    :    
//     name        :
//     date        :    
//                     (c)CGS
//     --------------------------------------------------------------------------------
BEGIN


       "SM_DATA_RESET"();                    //data block reset

       //actual hardware device configuration
       //------------------------------------
       "STA".ACT_DVC_CNF_BYTE_0  :=  DWORD_TO_BYTE("CNF".ACT_DVC_CNF);
       "STA".ACT_DVC_CNF_BYTE_1  :=  DWORD_TO_BYTE(SHR(IN:= "CNF".ACT_DVC_CNF, N:= 8));
       "STA".ACT_DVC_CNF_BYTE_2  :=  DWORD_TO_BYTE(SHR(IN:= "CNF".ACT_DVC_CNF, N:= 16));
       "STA".ACT_DVC_CNF_BYTE_3  :=  DWORD_TO_BYTE(SHR(IN:= "CNF".ACT_DVC_CNF, N:= 24));

       //presetting of main parameter variables
       //--------------------------------------
       "PAR_MAIN".DIA_MSR_PRD_NE         := 1.0;
       "PAR_MAIN".DIA_MSR_PRD_SH         := 1.0;
       "PAR_MAIN".DIA_MSR_PRD_BY         := 1.0;

       "PAR_MAIN".CH_GRAPH_TRANS_RAD     := 20.0;
       "PAR_MAIN".CH_GRAPH_BOTTOM_RAD    := 100.0;
       "PAR_MAIN".CH_GRAPH_INNER_DIA     := 100.0;

       "PAR_MAIN".PD_AMT_PRG_CYC         := 1.0;

       "PAR_MAIN".DI_TMP_DIPPING         := 900.0;

       "PAR_MAIN".BY_DIA_CTRL_ON_DLY     :=  30.0;
       "PAR_MAIN".BY_LEN_DIA_TMP_CTL_ON  := -1.0;

       "PAR_MAIN".RC_MAG_RATIO_CUR       :=  1.0;
       "PAR_MAIN".RC_PRS                 :=  3.0;

       "PAR_MAIN".MCONST_DIA_CAL_P1      := 100.0;
       "PAR_MAIN".MCONST_DIA_CAL_P2      := 100.0;
       "PAR_MAIN".MCONST_DIA_2_CAL_P1    := 100.0;
       "PAR_MAIN".MCONST_DIA_2_CAL_P2    := 100.0;

       "PAR_MAIN".MCONST_XT_LD_CELL_CAL  := 1.0;
       "PAR_MAIN".MCONST_MLT_LVL_CAL     := 1.0;

       "PAR_MAIN".ME_MAX_MLT_TMP         := 900.0;

       "KYA".SET_SEN_THR_P1              := 100.0;
       "KYA".SET_SEN_THR_P2              := 100.0;
       "KYA".SET_SEN_THR_P3              := 100.0;
       "KYA".SET_SEN_THR_P4              := 100.0;
       "KYA".SET_CAM_2_THR               := 100.0;

       "KYA".SET_SEN_CTR_X_P1            := 320.0;
       "KYA".SET_SEN_CTR_Y_P1            := 240.0;
       "KYA".SET_SEN_WDH_P1              := 200.0;
       "KYA".SET_SEN_HGT_P1              := 100.0;

       "KYA".SET_SEN_CTR_X_P2            := 320.0;
       "KYA".SET_SEN_CTR_Y_P2            := 240.0;
       "KYA".SET_SEN_OUT_RAD_P2          := 200.0;
       "KYA".SET_SEN_IN_RAD_P2           := 100.0;
       "KYA".SET_SEN_SEQ_STR_AGL_P2      := 62.0;
       "KYA".SET_SEN_SEQ_STP_AGL_P2      := 90.0;

       "KYA".SET_SEN_CTR_X_P3            := 320.0;
       "KYA".SET_SEN_CTR_Y_P3            := 240.0;
       "KYA".SET_SEN_WDH_P3              := 200.0;

       "KYA".SET_SEN_CTR_X_P4            := 320.0;
       "KYA".SET_SEN_CTR_Y_P4            := 240.0;
       "KYA".SET_SEN_WDH_P4              := 200.0;
       "KYA".SET_SEN_HGT_P4              := 100.0;

       "STA".ACT_STATE                   := 1;               //set state standby

       "STA".ACT_RCP_NAME                := '';              //initilisation of String variable
       "STA".ACT_INGOT_ID                := '';              //initilisation of String variable
       "STA".ACT_CRU_ID                  := '';              //initilisation of String variable
       "STA".ACT_CHARGE_ID               := '';              //initilisation of String variable
       "STA".USER_NAME                   := '';              //initilisation of String variable
       "STA".CARRIER_ID                  := '';              //initilisation of String variable
       "STA".AUX_INFO                    := '';              //initilisation of String variable
       "STA".AUX_COMMENT                 := '';              //initilistaion of String variable
       "STA".INGOT_ID_TIMEOUT            := 60;              //60 seconds timeout when CDP is not responding

       "KYA".SET_ROI_CTR_X_SCAM              := 600.0;
       "KYA".SET_ROI_CTR_Y_SCAM              := 700.0;
       "KYA".SET_ROI_HGT_SCAM                := 300.0;
       "KYA".SET_ROI_WDH_SCAM                := 400.0;

       "PAR_MAIN".MCONST_CF_TO_RAD_PT_SCAM   :=  0.0;                   //presetting
       "PAR_MAIN".MCONST_ANG_OF_PLX_SCAM     :=  0.0;                    //presetting
       "PAR_MAIN".MCONST_CAL_CF_SCAM         :=  0.0;                  //presetting
       "PAR_MAIN".MCONST_CAL_RAD_PT_SCAM     :=  0.0;                  //presetting
       "PAR_MAIN".MCONST_CAL_MLT_LVL_SCAM    :=  1.0;                    //presetting
       "PAR_SUB".SCAM_MLT_LVL_T1             :=  30.0;                   //presetting
       "PAR_SUB".CTR_X_SCAM_2_ADJ            :=  0.0;                    //presetting
       "PAR_SUB".CTR_Y_SCAM_2_ADJ            :=  0.0;                    //presetting
END_FUNCTION

FUNCTION "SM_FLT_RESET" : Void   // FC257, SCL
{ S7_Optimized_Access := 'FALSE' }
VERSION : 0.0
// --------------------------------------------------------------------------------
//     program     :    SM_FLT_RESET
//     description :    Reset alarms        
//     name        :    D. Bruess
//     date        :    11.11.99
// 
//     revision    :
//     name        :    G. Eibelsh鋟ser
//     date        :    1.12.99
//                     (c)CGS
//     --------------------------------------------------------------------------------
   VAR_INPUT
      linp : Word;
      ackn : Bool;
   END_VAR
   VAR_OUTPUT
      horn : Bool;
      icon : Bool;
   END_VAR
   VAR_IN_OUT
      lackn : Word;
      lnackn : Word;
   END_VAR
BEGIN

       IF (#linp <> #lackn) THEN                    //Verify if new faults are present

            //Acknowledged and reseted faults cleared in "not acknowledged fault list"                                      
            #lnackn := (((#linp XOR #lackn) AND #lackn) XOR #lnackn);   

            //Reseted faults cleared in "acknowledged fault list"                          
            #lackn := (((#linp XOR #lackn) AND #lackn) XOR #lackn);

            //Write new faults in "not acknowledged fault list"        
            #lnackn := ((#linp XOR #lnackn) OR #lnackn);

       END_IF;

      IF (#ackn = TRUE) THEN                       //If acknowledge button is activ 
            #lackn := #lnackn;                      //Transfer not ackn. faults to ackn. fault list
            #horn  := FALSE;                       //Reset Horn
       END_IF;

       IF (#lackn <> #lnackn) THEN                  //If not acknowledged faults are present
            #horn := TRUE;                         //Switch on horn
       ELSE #horn := FALSE;                        //otherwise disable horn
       END_IF;                                    

       IF (#lnackn <> 0) THEN                      //If faults in not acknowledge list are present
            #icon  := TRUE;                        //illuminate alarm icon on PC screen
       ELSE #icon  := FALSE;                       //reset alarm icon
       END_IF;
END_FUNCTION

FUNCTION "SM_CALL_FAULT_RESET" : Void   // FC258, SCL
{ S7_Optimized_Access := 'FALSE' }
VERSION : 0.0
// --------------------------------------------------------------------------------
//     program     :    SM_CALL_FAULT_RESET
//     description :    Call function to write acknowledged and not acknowledged 
//                      fault lists       
//     name        :    G. Eibelsh鋟ser
//     date        :    1.12.99
// 
//     revision    :
//     name        :
//     date        :    
//                     (c) CGS
//     --------------------------------------------------------------------------------
   VAR_TEMP
      alarmflag_0 : Bool;
      alarmflag_1 : Bool;
      alarmflag_2 : Bool;
      alarmflag_3 : Bool;
      alarmflag_4 : Bool;
      alarmflag_5 : Bool;
      alarmflag_6 : Bool;
      alarmflag_7 : Bool;
      alarmflag_8 : Bool;
      alarmflag_9 : Bool;
      alarmflag_10 : Bool;
      alarmflag_11 : Bool;
      alarmflag_12 : Bool;
      alarmflag_13 : Bool;
      alarmflag_14 : Bool;
      alarmflag_15 : Bool;
      alarmflag_16 : Bool;
      alarmflag_17 : Bool;
      alarmflag_18 : Bool;
      alarmflag_19 : Bool;
      alarmflag_20 : Bool;
      alarmflag_21 : Bool;
      alarmflag_22 : Bool;
      alarmflag_23 : Bool;
      alarmflag_24 : Bool;
      alarmflag_25 : Bool;
      alarmflag_26 : Bool;
      alarmflag_27 : Bool;
      alarmflag_28 : Bool;
      alarmflag_29 : Bool;
      alarmflag_30 : Bool;
      alarmflag_31 : Bool;
      alarmflag_32 : Bool;
      alarmflag_33 : Bool;
      alarmflag_34 : Bool;
      alarmflag_35 : Bool;
      alarmflag_36 : Bool;
      alarmflag_37 : Bool;
      alarmflag_38 : Bool;
      alarmflag_39 : Bool;
      alarmflag_40 : Bool;
      alarmflag_41 : Bool;
      alarmflag_42 : Bool;
      alarmflag_43 : Bool;
      alarmflag_44 : Bool;
      alarmflag_45 : Bool;
      alarmflag_46 : Bool;
      alarmflag_47 : Bool;
      alarmflag_48 : Bool;
      alarmflag_49 : Bool;
      alarmflag_50 : Bool;
      alarmflag_51 : Bool;
      alarmflag_52 : Bool;
      alarmflag_53 : Bool;
      alarmflag_54 : Bool;
      alarmflag_55 : Bool;
      alarmflag_56 : Bool;
      alarmflag_57 : Bool;
      alarmflag_58 : Bool;
      alarmflag_59 : Bool;
      alarmflag_60 : Bool;
      alarmflag_61 : Bool;
      alarmflag_62 : Bool;
      alarmflag_63 : Bool;
      hornflag : Bool;
      alarmicon_0 : Bool;
      alarmicon_1 : Bool;
      alarmicon_2 : Bool;
      alarmicon_3 : Bool;
      alarmicon_4 : Bool;
      alarmicon_5 : Bool;
      alarmicon_6 : Bool;
      alarmicon_7 : Bool;
      alarmicon_8 : Bool;
      alarmicon_9 : Bool;
      alarmicon_10 : Bool;
      alarmicon_11 : Bool;
      alarmicon_12 : Bool;
      alarmicon_13 : Bool;
      alarmicon_14 : Bool;
      alarmicon_15 : Bool;
      alarmicon_16 : Bool;
      alarmicon_17 : Bool;
      alarmicon_18 : Bool;
      alarmicon_19 : Bool;
      alarmicon_20 : Bool;
      alarmicon_21 : Bool;
      alarmicon_22 : Bool;
      alarmicon_23 : Bool;
      alarmicon_24 : Bool;
      alarmicon_25 : Bool;
      alarmicon_26 : Bool;
      alarmicon_27 : Bool;
      alarmicon_28 : Bool;
      alarmicon_29 : Bool;
      alarmicon_30 : Bool;
      alarmicon_31 : Bool;
      alarmicon_32 : Bool;
      alarmicon_33 : Bool;
      alarmicon_34 : Bool;
      alarmicon_35 : Bool;
      alarmicon_36 : Bool;
      alarmicon_37 : Bool;
      alarmicon_38 : Bool;
      alarmicon_39 : Bool;
      alarmicon_40 : Bool;
      alarmicon_41 : Bool;
      alarmicon_42 : Bool;
      alarmicon_43 : Bool;
      alarmicon_44 : Bool;
      alarmicon_45 : Bool;
      alarmicon_46 : Bool;
      alarmicon_47 : Bool;
      alarmicon_48 : Bool;
      alarmicon_49 : Bool;
      alarmicon_50 : Bool;
      alarmicon_51 : Bool;
      alarmicon_52 : Bool;
      alarmicon_53 : Bool;
      alarmicon_54 : Bool;
      alarmicon_55 : Bool;
      alarmicon_56 : Bool;
      alarmicon_57 : Bool;
      alarmicon_58 : Bool;
      alarmicon_59 : Bool;
      alarmicon_60 : Bool;
      alarmicon_61 : Bool;
      alarmicon_62 : Bool;
      alarmicon_63 : Bool;
   END_VAR
BEGIN


          "SM_FLT_RESET" (horn         => #alarmflag_0,
                        icon         => #alarmicon_0,
                        linp         := %DB142.%DBW0,
                        ackn         := "KYD".ALARM_ACKN,
                        lnackn       := "SM_FLT_NOT_ACKN".ALARM_WORD_0,    
                        lackn        := "SM_FLT_ACKN".ALARM_WORD_0);

          "SM_FLT_RESET" (horn         => #alarmflag_1,
                        icon         => #alarmicon_1,
                        linp         := %DB142.%DBW2,
                        ackn         := "KYD".ALARM_ACKN,
                        lnackn       := "SM_FLT_NOT_ACKN".ALARM_WORD_1,    
                        lackn        := "SM_FLT_ACKN".ALARM_WORD_1);

          "SM_FLT_RESET" (horn         => #alarmflag_2,
                        icon         => #alarmicon_2,
                        linp         := %DB142.%DBW4, 
                        ackn         := "KYD".ALARM_ACKN,
                        lnackn       := "SM_FLT_NOT_ACKN".ALARM_WORD_2,    
                        lackn        := "SM_FLT_ACKN".ALARM_WORD_2);

          "SM_FLT_RESET" (horn         => #alarmflag_3,
                        icon         => #alarmicon_3,
                        linp         := %DB142.%DBW6,
                        ackn         := "KYD".ALARM_ACKN,
                        lnackn       := "SM_FLT_NOT_ACKN".ALARM_WORD_3,    
                        lackn        := "SM_FLT_ACKN".ALARM_WORD_3);

          "SM_FLT_RESET" (horn         => #alarmflag_4,
                        icon         => #alarmicon_4,
                        linp         := %DB142.%DBW8, 
                        ackn         := "KYD".ALARM_ACKN,
                        lnackn       := "SM_FLT_NOT_ACKN".ALARM_WORD_4,    
                        lackn        := "SM_FLT_ACKN".ALARM_WORD_4);

          "SM_FLT_RESET" (horn         => #alarmflag_5,
                        icon         => #alarmicon_5,
                        linp         := %DB142.%DBW10,
                        ackn         := "KYD".ALARM_ACKN,
                        lnackn       := "SM_FLT_NOT_ACKN".ALARM_WORD_5,    
                        lackn        := "SM_FLT_ACKN".ALARM_WORD_5);

          "SM_FLT_RESET" (horn         => #alarmflag_6,
                        icon         => #alarmicon_6,
                        linp         := %DB142.%DBW12, 
                        ackn         := "KYD".ALARM_ACKN,
                        lnackn       := "SM_FLT_NOT_ACKN".ALARM_WORD_6,    
                        lackn        := "SM_FLT_ACKN".ALARM_WORD_6);

          "SM_FLT_RESET" (horn         => #alarmflag_7,
                        icon         => #alarmicon_7,
                        linp         := %DB142.%DBW14,
                        ackn         := "KYD".ALARM_ACKN,
                        lnackn       := "SM_FLT_NOT_ACKN".ALARM_WORD_7,    
                        lackn        := "SM_FLT_ACKN".ALARM_WORD_7);

          "SM_FLT_RESET" (horn         => #alarmflag_8,
                        icon         => #alarmicon_8,
                        linp         := %DB142.%DBW16,
                        ackn         := "KYD".ALARM_ACKN,
                        lnackn       := "SM_FLT_NOT_ACKN".ALARM_WORD_8,    
                        lackn        := "SM_FLT_ACKN".ALARM_WORD_8);

          "SM_FLT_RESET" (horn         => #alarmflag_9,
                        icon         => #alarmicon_9,
                        linp         := %DB142.%DBW18,
                        ackn         := "KYD".ALARM_ACKN,
                        lnackn       := "SM_FLT_NOT_ACKN".ALARM_WORD_9,    
                        lackn        := "SM_FLT_ACKN".ALARM_WORD_9);

          "SM_FLT_RESET" (horn         => #alarmflag_10,
                        icon         => #alarmicon_10,
                        linp         := %DB142.%DBW20, 
                        ackn         := "KYD".ALARM_ACKN,
                        lnackn       := "SM_FLT_NOT_ACKN".ALARM_WORD_10,    
                        lackn        := "SM_FLT_ACKN".ALARM_WORD_10);

          "SM_FLT_RESET" (horn         => #alarmflag_11,
                        icon         => #alarmicon_11,
                        linp         := %DB142.%DBW22,
                        ackn         := "KYD".ALARM_ACKN,
                        lnackn       := "SM_FLT_NOT_ACKN".ALARM_WORD_11,    
                        lackn        := "SM_FLT_ACKN".ALARM_WORD_11);

          "SM_FLT_RESET" (horn         => #alarmflag_12,
                        icon         => #alarmicon_12,
                        linp         := %DB142.%DBW24, 
                        ackn         := "KYD".ALARM_ACKN,
                        lnackn       := "SM_FLT_NOT_ACKN".ALARM_WORD_12,    
                        lackn        := "SM_FLT_ACKN".ALARM_WORD_12);

          "SM_FLT_RESET" (horn         => #alarmflag_13,
                        icon         => #alarmicon_13,
                        linp         := %DB142.%DBW26,
                        ackn         := "KYD".ALARM_ACKN,
                        lnackn       := "SM_FLT_NOT_ACKN".ALARM_WORD_13,    
                        lackn        := "SM_FLT_ACKN".ALARM_WORD_13);

          "SM_FLT_RESET" (horn         => #alarmflag_14,
                        icon         => #alarmicon_14,
                        linp         := %DB142.%DBW28, 
                        ackn         := "KYD".ALARM_ACKN,
                        lnackn       := "SM_FLT_NOT_ACKN".ALARM_WORD_14,    
                        lackn        := "SM_FLT_ACKN".ALARM_WORD_14);

          "SM_FLT_RESET" (horn         => #alarmflag_15,
                        icon         => #alarmicon_15,
                        linp         := %DB142.%DBW30,
                        ackn         := "KYD".ALARM_ACKN,
                        lnackn       := "SM_FLT_NOT_ACKN".ALARM_WORD_15,    
                        lackn        := "SM_FLT_ACKN".ALARM_WORD_15);

          "SM_FLT_RESET" (horn         => #alarmflag_16,
                        icon         => #alarmicon_16,
                        linp         := %DB142.%DBW32,
                        ackn         := "KYD".ALARM_ACKN,
                        lnackn       := "SM_FLT_NOT_ACKN".ALARM_WORD_16,    
                        lackn        := "SM_FLT_ACKN".ALARM_WORD_16);

          "SM_FLT_RESET" (horn         => #alarmflag_17,
                        icon         => #alarmicon_17,
                        linp         := %DB142.%DBW34,
                        ackn         := "KYD".ALARM_ACKN,
                        lnackn       := "SM_FLT_NOT_ACKN".ALARM_WORD_17,    
                        lackn        := "SM_FLT_ACKN".ALARM_WORD_17);

          "SM_FLT_RESET" (horn         => #alarmflag_18,
                        icon         => #alarmicon_18,
                        linp         := %DB142.%DBW36,
                        ackn         := "KYD".ALARM_ACKN,
                        lnackn       := "SM_FLT_NOT_ACKN".ALARM_WORD_18,    
                        lackn        := "SM_FLT_ACKN".ALARM_WORD_18);

          "SM_FLT_RESET" (horn         => #alarmflag_19,
                        icon         => #alarmicon_19,
                        linp         := %DB142.%DBW38,
                        ackn         := "KYD".ALARM_ACKN,
                        lnackn       := "SM_FLT_NOT_ACKN".ALARM_WORD_19,    
                        lackn        := "SM_FLT_ACKN".ALARM_WORD_19);

          "SM_FLT_RESET" (horn         => #alarmflag_20,
                        icon         => #alarmicon_20,
                        linp         := %DB142.%DBW40,
                        ackn         := "KYD".ALARM_ACKN,
                        lnackn       := "SM_FLT_NOT_ACKN".ALARM_WORD_20,    
                        lackn        := "SM_FLT_ACKN".ALARM_WORD_20);

          "SM_FLT_RESET" (horn         => #alarmflag_21,
                        icon         => #alarmicon_21,
                        linp         := %DB142.%DBW42,
                        ackn         := "KYD".ALARM_ACKN,
                        lnackn       := "SM_FLT_NOT_ACKN".ALARM_WORD_21,    
                        lackn        := "SM_FLT_ACKN".ALARM_WORD_21);

          "SM_FLT_RESET" (horn         => #alarmflag_22,
                        icon         => #alarmicon_22,
                        linp         := %DB142.%DBW44,
                        ackn         := "KYD".ALARM_ACKN,
                        lnackn       := "SM_FLT_NOT_ACKN".ALARM_WORD_22,    
                        lackn        := "SM_FLT_ACKN".ALARM_WORD_22);

          "SM_FLT_RESET" (horn         => #alarmflag_23,
                        icon         => #alarmicon_23,
                        linp         := %DB142.%DBW46,
                        ackn         := "KYD".ALARM_ACKN,
                        lnackn       := "SM_FLT_NOT_ACKN".ALARM_WORD_23,    
                        lackn        := "SM_FLT_ACKN".ALARM_WORD_23);

          "SM_FLT_RESET" (horn         => #alarmflag_24,
                        icon         => #alarmicon_24,
                        linp         := %DB142.%DBW48,
                        ackn         := "KYD".ALARM_ACKN,
                        lnackn       := "SM_FLT_NOT_ACKN".ALARM_WORD_24,    
                        lackn        := "SM_FLT_ACKN".ALARM_WORD_24);

          "SM_FLT_RESET" (horn         => #alarmflag_25,
                        icon         => #alarmicon_25,
                        linp         := %DB142.%DBW50,
                        ackn         := "KYD".ALARM_ACKN,
                        lnackn       := "SM_FLT_NOT_ACKN".ALARM_WORD_25,    
                        lackn        := "SM_FLT_ACKN".ALARM_WORD_25);

          "SM_FLT_RESET" (horn         => #alarmflag_26,
                        icon         => #alarmicon_26,
                        linp         := %DB142.%DBW52,
                        ackn         := "KYD".ALARM_ACKN,
                        lnackn       := "SM_FLT_NOT_ACKN".ALARM_WORD_26,    
                        lackn        := "SM_FLT_ACKN".ALARM_WORD_26);

          "SM_FLT_RESET" (horn         => #alarmflag_27,
                        icon         => #alarmicon_27,
                        linp         := %DB142.%DBW54,
                        ackn         := "KYD".ALARM_ACKN,
                        lnackn       := "SM_FLT_NOT_ACKN".ALARM_WORD_27,    
                        lackn        := "SM_FLT_ACKN".ALARM_WORD_27);

          "SM_FLT_RESET" (horn         => #alarmflag_28,
                        icon         => #alarmicon_28,
                        linp         := %DB142.%DBW56,
                        ackn         := "KYD".ALARM_ACKN,
                        lnackn       := "SM_FLT_NOT_ACKN".ALARM_WORD_28,    
                        lackn        := "SM_FLT_ACKN".ALARM_WORD_28);

          "SM_FLT_RESET" (horn         => #alarmflag_29,
                        icon         => #alarmicon_29,
                        linp         := %DB142.%DBW58,
                        ackn         := "KYD".ALARM_ACKN,
                        lnackn       := "SM_FLT_NOT_ACKN".ALARM_WORD_29,    
                        lackn        := "SM_FLT_ACKN".ALARM_WORD_29);

          "SM_FLT_RESET" (horn         => #alarmflag_30,
                        icon         => #alarmicon_30,
                        linp         := %DB142.%DBW60,
                        ackn         := "KYD".ALARM_ACKN,
                        lnackn       := "SM_FLT_NOT_ACKN".ALARM_WORD_30,    
                        lackn        := "SM_FLT_ACKN".ALARM_WORD_30);

           "SM_FLT_RESET" (horn         => #alarmflag_31,
                        icon         => #alarmicon_31,
                        linp         := %DB142.%DBW62,
                        ackn         := "KYD".ALARM_ACKN,
                        lnackn       := "SM_FLT_NOT_ACKN".ALARM_WORD_31,    
                        lackn        := "SM_FLT_ACKN".ALARM_WORD_31);

          "SM_FLT_RESET" (horn         => #alarmflag_32,
                        icon         => #alarmicon_32,
                        linp         := %DB142.%DBW64,
                        ackn         := "KYD".ALARM_ACKN,
                        lnackn       := "SM_FLT_NOT_ACKN".ALARM_WORD_32,    
                        lackn        := "SM_FLT_ACKN".ALARM_WORD_32);

          "SM_FLT_RESET" (horn         => #alarmflag_33,
                        icon         => #alarmicon_33,
                        linp         := %DB142.%DBW66,
                        ackn         := "KYD".ALARM_ACKN,
                        lnackn       := "SM_FLT_NOT_ACKN".ALARM_WORD_33,    
                        lackn        := "SM_FLT_ACKN".ALARM_WORD_33);

          "SM_FLT_RESET" (horn         => #alarmflag_34,
                        icon         => #alarmicon_34,
                        linp         := %DB142.%DBW68, 
                        ackn         := "KYD".ALARM_ACKN,
                        lnackn       := "SM_FLT_NOT_ACKN".ALARM_WORD_34,    
                        lackn        := "SM_FLT_ACKN".ALARM_WORD_34);

          "SM_FLT_RESET" (horn         => #alarmflag_35,
                        icon         => #alarmicon_35,
                        linp         := %DB142.%DBW70,
                        ackn         := "KYD".ALARM_ACKN,
                        lnackn       := "SM_FLT_NOT_ACKN".ALARM_WORD_35,    
                        lackn        := "SM_FLT_ACKN".ALARM_WORD_35);

          "SM_FLT_RESET" (horn         => #alarmflag_36,
                        icon         => #alarmicon_36,
                        linp         := %DB142.%DBW72, 
                        ackn         := "KYD".ALARM_ACKN,
                        lnackn       := "SM_FLT_NOT_ACKN".ALARM_WORD_36,    
                        lackn        := "SM_FLT_ACKN".ALARM_WORD_36);

          "SM_FLT_RESET" (horn         => #alarmflag_37,
                        icon         => #alarmicon_37,
                        linp         := %DB142.%DBW74,
                        ackn         := "KYD".ALARM_ACKN,
                        lnackn       := "SM_FLT_NOT_ACKN".ALARM_WORD_37,    
                        lackn        := "SM_FLT_ACKN".ALARM_WORD_37);

          "SM_FLT_RESET" (horn         => #alarmflag_38,
                        icon         => #alarmicon_38,
                        linp         := %DB142.%DBW76, 
                        ackn         := "KYD".ALARM_ACKN,
                        lnackn       := "SM_FLT_NOT_ACKN".ALARM_WORD_38,    
                        lackn        := "SM_FLT_ACKN".ALARM_WORD_38);

          "SM_FLT_RESET" (horn         => #alarmflag_39,
                        icon         => #alarmicon_39,
                        linp         := %DB142.%DBW78,
                        ackn         := "KYD".ALARM_ACKN,
                        lnackn       := "SM_FLT_NOT_ACKN".ALARM_WORD_39,    
                        lackn        := "SM_FLT_ACKN".ALARM_WORD_39);

          "SM_FLT_RESET" (horn         => #alarmflag_40,
                        icon         => #alarmicon_40,
                        linp         := %DB142.%DBW80,
                        ackn         := "KYD".ALARM_ACKN,
                        lnackn       := "SM_FLT_NOT_ACKN".ALARM_WORD_40,    
                        lackn        := "SM_FLT_ACKN".ALARM_WORD_40);

          "SM_FLT_RESET" (horn         => #alarmflag_41,
                        icon         => #alarmicon_41,
                        linp         := %DB142.%DBW82,
                        ackn         := "KYD".ALARM_ACKN,
                        lnackn       := "SM_FLT_NOT_ACKN".ALARM_WORD_41,    
                        lackn        := "SM_FLT_ACKN".ALARM_WORD_41);

          "SM_FLT_RESET" (horn         => #alarmflag_42,
                        icon         => #alarmicon_42,
                        linp         := %DB142.%DBW84, 
                        ackn         := "KYD".ALARM_ACKN,
                        lnackn       := "SM_FLT_NOT_ACKN".ALARM_WORD_42,    
                        lackn        := "SM_FLT_ACKN".ALARM_WORD_42);

          "SM_FLT_RESET" (horn         => #alarmflag_43,
                        icon         => #alarmicon_43,
                        linp         := %DB142.%DBW86,
                        ackn         := "KYD".ALARM_ACKN,
                        lnackn       := "SM_FLT_NOT_ACKN".ALARM_WORD_43,    
                        lackn        := "SM_FLT_ACKN".ALARM_WORD_43);

          "SM_FLT_RESET" (horn         => #alarmflag_44,
                        icon         => #alarmicon_44,
                        linp         := %DB142.%DBW88, 
                        ackn         := "KYD".ALARM_ACKN,
                        lnackn       := "SM_FLT_NOT_ACKN".ALARM_WORD_44,    
                        lackn        := "SM_FLT_ACKN".ALARM_WORD_44);

          "SM_FLT_RESET" (horn         => #alarmflag_45,
                        icon         => #alarmicon_45,
                        linp         := %DB142.%DBW90,
                        ackn         := "KYD".ALARM_ACKN,
                        lnackn       := "SM_FLT_NOT_ACKN".ALARM_WORD_45,    
                        lackn        := "SM_FLT_ACKN".ALARM_WORD_45);

          "SM_FLT_RESET" (horn         => #alarmflag_46,
                        icon         => #alarmicon_46,
                        linp         := %DB142.%DBW92, 
                        ackn         := "KYD".ALARM_ACKN,
                        lnackn       := "SM_FLT_NOT_ACKN".ALARM_WORD_46,    
                        lackn        := "SM_FLT_ACKN".ALARM_WORD_46);

          "SM_FLT_RESET" (horn         => #alarmflag_47,
                        icon         => #alarmicon_47,
                        linp         := %DB142.%DBW94,
                        ackn         := "KYD".ALARM_ACKN,
                        lnackn       := "SM_FLT_NOT_ACKN".ALARM_WORD_47,    
                        lackn        := "SM_FLT_ACKN".ALARM_WORD_47);

          "SM_FLT_RESET" (horn         => #alarmflag_48,
                        icon         => #alarmicon_48,
                        linp         := %DB142.%DBW96,
                        ackn         := "KYD".ALARM_ACKN,
                        lnackn       := "SM_FLT_NOT_ACKN".ALARM_WORD_48,    
                        lackn        := "SM_FLT_ACKN".ALARM_WORD_48);

          "SM_FLT_RESET" (horn         => #alarmflag_49,
                        icon         => #alarmicon_49,
                        linp         := %DB142.%DBW98,
                        ackn         := "KYD".ALARM_ACKN,
                        lnackn       := "SM_FLT_NOT_ACKN".ALARM_WORD_49,    
                        lackn        := "SM_FLT_ACKN".ALARM_WORD_49);

          "SM_FLT_RESET" (horn         => #alarmflag_50,
                        icon         => #alarmicon_50,
                        linp         := %DB142.%DBW100,
                        ackn         := "KYD".ALARM_ACKN,
                        lnackn       := "SM_FLT_NOT_ACKN".ALARM_WORD_50,    
                        lackn        := "SM_FLT_ACKN".ALARM_WORD_50);

          "SM_FLT_RESET" (horn         => #alarmflag_51,
                        icon         => #alarmicon_51,
                        linp         := %DB142.%DBW102,
                        ackn         := "KYD".ALARM_ACKN,
                        lnackn       := "SM_FLT_NOT_ACKN".ALARM_WORD_51,    
                        lackn        := "SM_FLT_ACKN".ALARM_WORD_51);

          "SM_FLT_RESET" (horn         => #alarmflag_52,
                        icon         => #alarmicon_52,
                        linp         := %DB142.%DBW104,
                        ackn         := "KYD".ALARM_ACKN,
                        lnackn       := "SM_FLT_NOT_ACKN".ALARM_WORD_52,    
                        lackn        := "SM_FLT_ACKN".ALARM_WORD_52);

          "SM_FLT_RESET" (horn         => #alarmflag_53,
                        icon         => #alarmicon_53,
                        linp         := %DB142.%DBW106,
                        ackn         := "KYD".ALARM_ACKN,
                        lnackn       := "SM_FLT_NOT_ACKN".ALARM_WORD_53,    
                        lackn        := "SM_FLT_ACKN".ALARM_WORD_53);

          "SM_FLT_RESET" (horn         => #alarmflag_54,
                        icon         => #alarmicon_54,
                        linp         := %DB142.%DBW108,
                        ackn         := "KYD".ALARM_ACKN,
                        lnackn       := "SM_FLT_NOT_ACKN".ALARM_WORD_54,    
                        lackn        := "SM_FLT_ACKN".ALARM_WORD_54);

          "SM_FLT_RESET" (horn         => #alarmflag_55,
                        icon         => #alarmicon_55,
                        linp         := %DB142.%DBW110,
                        ackn         := "KYD".ALARM_ACKN,
                        lnackn       := "SM_FLT_NOT_ACKN".ALARM_WORD_55,    
                        lackn        := "SM_FLT_ACKN".ALARM_WORD_55);

          "SM_FLT_RESET" (horn         => #alarmflag_56,
                        icon         => #alarmicon_56,
                        linp         := %DB142.%DBW112,
                        ackn         := "KYD".ALARM_ACKN,
                        lnackn       := "SM_FLT_NOT_ACKN".ALARM_WORD_56,    
                        lackn        := "SM_FLT_ACKN".ALARM_WORD_56);

          "SM_FLT_RESET" (horn         => #alarmflag_57,
                        icon         => #alarmicon_57,
                        linp         := %DB142.%DBW114,
                        ackn         := "KYD".ALARM_ACKN,
                        lnackn       := "SM_FLT_NOT_ACKN".ALARM_WORD_57,    
                        lackn        := "SM_FLT_ACKN".ALARM_WORD_57);

          "SM_FLT_RESET" (horn         => #alarmflag_58,
                        icon         => #alarmicon_58,
                        linp         := %DB142.%DBW116,
                        ackn         := "KYD".ALARM_ACKN,
                        lnackn       := "SM_FLT_NOT_ACKN".ALARM_WORD_58,    
                        lackn        := "SM_FLT_ACKN".ALARM_WORD_58);

          "SM_FLT_RESET" (horn         => #alarmflag_59,
                        icon         => #alarmicon_59,
                        linp         := %DB142.%DBW118,
                        ackn         := "KYD".ALARM_ACKN,
                        lnackn       := "SM_FLT_NOT_ACKN".ALARM_WORD_59,    
                        lackn        := "SM_FLT_ACKN".ALARM_WORD_59);

          "SM_FLT_RESET" (horn         => #alarmflag_60,
                        icon         => #alarmicon_60,
                        linp         := %DB142.%DBW120,
                        ackn         := "KYD".ALARM_ACKN,
                        lnackn       := "SM_FLT_NOT_ACKN".ALARM_WORD_60,    
                        lackn        := "SM_FLT_ACKN".ALARM_WORD_60);

          "SM_FLT_RESET" (horn         => #alarmflag_61,
                        icon         => #alarmicon_61,
                        linp         := %DB142.%DBW122,
                        ackn         := "KYD".ALARM_ACKN,
                        lnackn       := "SM_FLT_NOT_ACKN".ALARM_WORD_61,    
                        lackn        := "SM_FLT_ACKN".ALARM_WORD_61);

          "SM_FLT_RESET" (horn         => #alarmflag_62,
                        icon         => #alarmicon_62,
                        linp         := %DB142.%DBW124,
                        ackn         := "KYD".ALARM_ACKN,
                        lnackn       := "SM_FLT_NOT_ACKN".ALARM_WORD_62,    
                        lackn        := "SM_FLT_ACKN".ALARM_WORD_62);

          "SM_FLT_RESET" (horn         => #alarmflag_63,
                        icon         => #alarmicon_63,
                        linp         := %DB142.%DBW126,
                        ackn         := "KYD".ALARM_ACKN,
                        lnackn       := "SM_FLT_NOT_ACKN".ALARM_WORD_63,    
                        lackn        := "SM_FLT_ACKN".ALARM_WORD_63);


       //collect fault signals from all alarm words 
       //------------------------------------------ 
       #hornflag := #alarmflag_0     OR 
                   #alarmflag_1     OR 
                   #alarmflag_2     OR 
                   #alarmflag_3     OR 
                   #alarmflag_4     OR 
                   #alarmflag_5     OR
                   #alarmflag_6     OR
                   #alarmflag_7     OR
                   #alarmflag_8     OR 
                   #alarmflag_9     OR 
                   #alarmflag_10    OR 
                   #alarmflag_11    OR 
                   #alarmflag_12    OR 
                   #alarmflag_13    OR
                   #alarmflag_14    OR
                   #alarmflag_15    OR 
                   #alarmflag_16    OR 
                   #alarmflag_17    OR 
                   #alarmflag_18    OR 
                   #alarmflag_19    OR 
                   #alarmflag_20    OR 
                   #alarmflag_21    OR
                   #alarmflag_22    OR
                   #alarmflag_23    OR
                   #alarmflag_24    OR 
                   #alarmflag_25    OR 
                   #alarmflag_26    OR 
                   #alarmflag_27    OR 
                   #alarmflag_28    OR 
                   #alarmflag_29    OR
                   #alarmflag_30    OR
                   #alarmflag_31    OR
                   #alarmflag_32    OR 
                   #alarmflag_33    OR 
                   #alarmflag_34    OR 
                   #alarmflag_35    OR 
                   #alarmflag_36    OR 
                   #alarmflag_37    OR
                   #alarmflag_38    OR
                   #alarmflag_39    OR
                   #alarmflag_40    OR 
                   #alarmflag_41    OR 
                   #alarmflag_42    OR 
                   #alarmflag_43    OR 
                   #alarmflag_44    OR 
                   #alarmflag_45    OR
                   #alarmflag_46    OR
                   #alarmflag_47    OR 
                   #alarmflag_48    OR 
                   #alarmflag_49    OR 
                   #alarmflag_50    OR 
                   #alarmflag_51    OR 
                   #alarmflag_52    OR 
                   #alarmflag_53    OR
                   #alarmflag_54    OR
                   #alarmflag_55    OR
                   #alarmflag_56    OR 
                   #alarmflag_57    OR 
                   #alarmflag_58    OR 
                   #alarmflag_59    OR 
                   #alarmflag_60    OR 
                   #alarmflag_61    OR
                   #alarmflag_62    OR
                   #alarmflag_63;

       //set output of acustic and optical alarm signal
       //---------------------------------------------- 
       "PDO".HOR_OPP_K2     :=  ((#hornflag OR "DV".HOR_OPP) AND "APC".BLK) OR          //alarm horn active
                              (NOT #hornflag AND "BM_OP_CALL_DB".OP_CALL_ALM AND "BM_OP_CALL_DB".OP_CALL_ALM) OR
                              (NOT #hornflag AND ("BM_OP_CALL_DB".OP_CALL_ALM OR "DV".AUTO_OP_CALL) AND "BM_OP_CALL_DB".OP_CALL_ALM);                            
       "PDO".HOR_OPP_K8     :=  "PDO".HOR_OPP_K2;
       "PDO".HOR_OPP_K9     :=  "PDO".HOR_OPP_K2;

       "PDO".LMP_RD_K2      :=  ((#hornflag OR "DV".HOR_OPP) AND "APC".BLK) OR 
                              (NOT #hornflag AND "LT".ALARM);
       "PDO".LMP_RD_K8      :=  "PDO".LMP_RD_K2;
       "PDO".LMP_RD_K9      :=  "PDO".LMP_RD_K2;

       "PDO".LMP_YE_K2      :=  "PDO".LMP_MAG_ACTIVE OR "DV".LMP_OR;
       "PDO".LMP_YE_K8      :=  "PDO".LMP_YE_K2;
       "PDO".LMP_YE_K9      :=  "PDO".LMP_YE_K2;

       "PDO".LMP_GN_K2      :=  NOT("LT".MOD_SERVICE OR "LT".MOD_SEMI_AUTO);
       "PDO".LMP_GN_K8      :=  "PDO".LMP_GN_K2;
       "PDO".LMP_GN_K9      :=  "PDO".LMP_GN_K2;

       "PDO".LMP_BU_K2      :=  "APC".AUTOMATIC;
       "PDO".LMP_BU_K8      :=  "PDO".LMP_BU_K2;
       "PDO".LMP_BU_K9      :=  "PDO".LMP_BU_K2;

       //set light variable when not acknowledged alarms are active
       //----------------------------------------------------------
       "LT".NOT_ACKN_ALM :=  #hornflag;   //only used in PMS

       //set variable of alarm icon on pc screen
       //---------------------------------------
       "LT".ALARM := #alarmicon_0     OR 
                   #alarmicon_1     OR 
                   #alarmicon_2     OR 
                   #alarmicon_3     OR 
                   #alarmicon_4     OR 
                   #alarmicon_5     OR
                   #alarmicon_6     OR
                   #alarmicon_7     OR
                   #alarmicon_8     OR 
                   #alarmicon_9     OR 
                   #alarmicon_10    OR 
                   #alarmicon_11    OR 
                   #alarmicon_12    OR 
                   #alarmicon_13    OR
                   #alarmicon_14    OR
                   #alarmicon_15    OR
                   #alarmicon_16    OR 
                   #alarmicon_17    OR 
                   #alarmicon_18    OR 
                   #alarmicon_19    OR 
                   #alarmicon_20    OR 
                   #alarmicon_21    OR
                   #alarmicon_22    OR
                   #alarmicon_23    OR
                   #alarmicon_24    OR 
                   #alarmicon_25    OR 
                   #alarmicon_26    OR 
                   #alarmicon_27    OR 
                   #alarmicon_28    OR 
                   #alarmicon_29    OR
                   #alarmicon_30    OR
                   #alarmicon_31    OR 
                   #alarmicon_32    OR 
                   #alarmicon_33    OR 
                   #alarmicon_34    OR 
                   #alarmicon_35    OR 
                   #alarmicon_36    OR 
                   #alarmicon_37    OR
                   #alarmicon_38    OR
                   #alarmicon_39    OR
                   #alarmicon_40    OR 
                   #alarmicon_41    OR 
                   #alarmicon_42    OR 
                   #alarmicon_43    OR 
                   #alarmicon_44    OR 
                   #alarmicon_45    OR
                   #alarmicon_46    OR
                   #alarmicon_47    OR 
                   #alarmicon_48    OR 
                   #alarmicon_49    OR 
                   #alarmicon_50    OR 
                   #alarmicon_51    OR 
                   #alarmicon_52    OR 
                   #alarmicon_53    OR
                   #alarmicon_54    OR
                   #alarmicon_55    OR
                   #alarmicon_56    OR 
                   #alarmicon_57    OR 
                   #alarmicon_58    OR 
                   #alarmicon_59    OR 
                   #alarmicon_60    OR 
                   #alarmicon_61    OR
                   #alarmicon_62    OR
                   #alarmicon_63;
END_FUNCTION

FUNCTION "SM_FLT_SETP_DEV_DLY" : Void   // FC259, SCL
{ S7_Optimized_Access := 'FALSE' }
VERSION : 0.0
// --------------------------------------------------------------------------------
//     program     :    SM_FLT_SETP_DEV_DLY
//     description :    Check actual deviation from setpoint       
//     name        :    G. Eibelsh鋟ser
//     date        :    04.02.00
// 
//     revision    :
//     name        :
//     date        :    
//                     (c) CGS
//     --------------------------------------------------------------------------------
   VAR_INPUT
      act_value : Real;
      set_value : Real;
      max_dev : Real;
      delay_time : Real;
      enable : Bool;
   END_VAR
   VAR_OUTPUT
      fault : Bool;
   END_VAR
BEGIN


   IF (#enable) AND #delay_time    <=    999.0    THEN    //max. delay time is 999 sec., 
                                                        //larger time disables deviation control
       IF     #set_value - #max_dev    <=    #act_value    AND
              #set_value + #max_dev    >=    #act_value    THEN

              #fault        :=    false;           
       ELSE   #fault        :=    true;

       END_IF;
   ELSE
       #fault    :=    false;    

   END_IF;
END_FUNCTION

FUNCTION "SM_FLT_SET_ALM" : Void   // FC260, SCL
{ S7_Optimized_Access := 'FALSE' }
VERSION : 0.0
BEGIN

      // Emergency off
      //------------------
      "FLT".EMO         := NOT "PDI".EMO;
      "FLT".EMS_HDL_DRV := NOT "PDI".EMS;

      //breakers and fuses
      //------------------
      "FLT".CB_FLT_DC24V      := NOT "PDI".CB_FLT_DC24V_K2 OR NOT "PDI".CB_FLT_DC24V_K5;
      "FLT".CB_FLT_AC230V     := NOT "PDI".CB_FLT_AC230V;
      "FLT".CB_FLT_AC400V     := NOT "PDI".CB_FLT_AC400V_K2 OR NOT "PDI".CB_FLT_AC400V_K2;
      "FLT".CB_FLT_DRV        := NOT "PDI".CB_FLT_AC400V_K8 OR NOT "PDI".CB_FLT_DC24V_K8;

      //24V UPS alarms
      //--------------
      "FLT".UPS_24V_ALM       := NOT "PDI".UPS_24V_ALM;
      "FLT".UPS_24V_SPL_MIS   := "PDI".UPS_24V_NRM;
      "DV".MAIN_SWITCH_ON     := NOT "PDI".UPS_24V_NRM;
END_FUNCTION

FUNCTION "SM_POS_EDGE" : Void   // FC262, SCL
{ S7_Optimized_Access := 'FALSE' }
VERSION : 0.0
// -----------------------------------------------------------------------------------
//     program     :   SM_POS_EDGE
//     description :   each positive edge detection of an input flag inverts 
//                     the output flag
//     name        :   G. Eibelsh鋟ser
//     date        :   07.04.2016
// 
//     
//                     (c)PVA CGS GmbH       
// -----------------------------------------------------------------------------------
   VAR_INPUT
      input : Bool;
   END_VAR
   VAR_IN_OUT
      busy : Bool;
      output : Bool;
   END_VAR
BEGIN

       //detect positive edge of input flag
       //----------------------------------
       IF #input AND NOT #busy THEN
           //invert output flag 
           //------------------
           IF #output THEN
               #output  :=  false;
           ELSE
               #output  :=  true;
           END_IF;
       END_IF;
       //store status of input flag
       //--------------------------
       #busy    :=  #input;
END_FUNCTION

FUNCTION "SM_NEG_EDGE" : Void   // FC263, SCL
{ S7_Optimized_Access := 'FALSE' }
VERSION : 0.0
// -----------------------------------------------------------------------------------
//     program     :   SM_NEG_EDGE
//     description :   each negative edge detection of an input flag inverts 
//                     the output flag
//     name        :   G. Eibelsh鋟ser
//     date        :   07.04.2016
// 
//     
//                     (c)PVA CGS GmbH       
// -----------------------------------------------------------------------------------
   VAR_INPUT
      input : Bool;
   END_VAR
   VAR_IN_OUT
      busy : Bool;
      output : Bool;
   END_VAR
BEGIN

       //detect negative edge of input flag
       //----------------------------------
       IF NOT #input AND #busy THEN
           //invert output flag 
           //------------------
           IF #output THEN
               #output  :=  false;
           ELSE
               #output  :=  true;
           END_IF;

       END_IF;
       //store status of input flag
       //--------------------------
       #busy    :=  #input;
END_FUNCTION

FUNCTION "SM_DATA_RESET" : Void   // FC264, SCL
{ S7_Optimized_Access := 'FALSE' }
VERSION : 0.0
// --------------------------------------------------------------------------------
//     program     :    SM_DATA_RESET
//     description :    reset variables data blocks       
//     name        :    K. Kalkowski
//     date        :    04.11.98
// 
//     revision    :    data blocks included:
//                             PAR_MAG_RATIO_CUR
//                             PAR_GAS_SUM_FLW
//                             PAR_TME
//                             SM_FLT_ACKN
//                             SM_FLT_NOT_ACKN
//                             STA
//                             CM_LOOP_PRS_DB
//                             CM_LOOP_DIA_DB
//                             CM_LOOP_HTR_1_DB
//                             CM_LOOP_HTR_2_DB
//                             CM_LOOP_AVG_SPD_DB
//                             CM_LOOP_MLT_TMP_DB
//                             CM_LOOP_GRW_RTE_DB
//                             CM_LOOP_MLT_LVL_DB
//                             CM_LOOP_PRS_DB
//                             CRUC
//                             AM_PRS_CTRL_DB
//                             AM_XT_DRV_MOVE_DB
//                             AM_CR_DRV_MOVE_DB
//                             AM_ID_DB
//                             AM_ME_DB
//                             AM_DI_DB
//                             AM_NE_DB
//                             AM_SH_DB
//                             AM_BY_DB
//                             AM_EC_DB
//                             AM_SD_DB
//                             AM_RE_DB
//                             BM_CALL_DRV_DB
//                             BM_CALL_PS_DB
//                             BM_CAM_CONTROL_DB
//     name        :    D.Bruess
//     date        :    04.02.00
//     
//     revision    :    data blocks included:
//                             SY
//     name        :    D.Bruess
//     date        :    07.03.00
// 
//     revision    :    data blocks included:
//                             PM_DVC_DRV_CTRL_DB
//                             PM_DVC_PS_CTRL_DB
//     name        :    D.Bruess
//     date        :    09.03.00
// 
//     name        :    H.Paki
//     date        :    17.03.00    **hp .....
// 
//     
//     name        :    G. Eibelsh鋟ser
//     date        :    13.07.00   
//     revision    :    data block included:
//                             BM_DRV_CAL_DB       
//                             
//     name        :    G. Eibelsh鋟ser
//     date        :    19.03.01   
//     revision    :    data block included:
//                             PAR_SUB       
//                             
//     name        :    M.Lech
//     date        :    11.05.01   
//     revision    :    data block included:
//                             BM_DRV_WHILE_LRT       
// 
//     name        :    M.Lech
//     date        :    13.02.02   
//     revision    :    data blocks included:
//                             BM_FDR_DB
//                             BM_FDR_MOVE_HOME_DB
//                             BM_FDR_SEQ_DB
//                             BM_FDR_LEAK_TST
//                             
//     name        :    M.Lech
//     date        :    20.02.03   
//     revision    :    data block included:
//                             BM_SEED_TMP_CTL_DB
//  
// 
//                     (c)CGS
//     --------------------------------------------------------------------------------
   VAR_TEMP
      return_sfc21 : Int;   // return value sfc21
      fill_value_0 : DWord;   // fill value 0
      fill_value_1 : DWord;   // fill value 1
      fill_value_2 : DWord;   // fill value 2
   END_VAR
BEGIN

       #fill_value_0 := 16#00000000;    // =>> float 0.0
       #fill_value_1 := 16#3F800000;    // =>> float 1.0
       #fill_value_2 := 16#40400000;    // =>> float 3.0


       #return_sfc21 := FILL(BVAL := #fill_value_0, BLK    =>  "SY");
       //parameter data blocks
       //---------------------
       #return_sfc21 := FILL(BVAL := #fill_value_0, BLK    =>  "PAR_SUB");    
       #return_sfc21 := FILL(BVAL := #fill_value_0, BLK    =>  "PAR_MAIN");
       #return_sfc21 := FILL(BVAL := #fill_value_0, BLK    =>  "PAR_XT_SPD");
       #return_sfc21 := FILL(BVAL := #fill_value_0, BLK    =>  "PAR_XT_ROT");
       #return_sfc21 := FILL(BVAL := #fill_value_0, BLK    =>  "PAR_XT_POS");
       #return_sfc21 := FILL(BVAL := #fill_value_0, BLK    =>  "PAR_CR_SPD");
       #return_sfc21 := FILL(BVAL := #fill_value_0, BLK    =>  "PAR_CR_ROT");
       #return_sfc21 := FILL(BVAL := #fill_value_0, BLK    =>  "PAR_CR_POS");
       #return_sfc21 := FILL(BVAL := #fill_value_0, BLK    =>  "PAR_CRSPD_COEFF");
       #return_sfc21 := FILL(BVAL := #fill_value_0, BLK    =>  "PAR_CR_ROT_ON_TME");
       #return_sfc21 := FILL(BVAL := #fill_value_0, BLK    =>  "PAR_CR_ROT_OFF_TME");
       #return_sfc21 := FILL(BVAL := #fill_value_0, BLK    =>  "PAR_CR_ROT_OFFSET");
       #return_sfc21 := FILL(BVAL := #fill_value_0, BLK    =>  "PAR_HTR_1_PWR");
       #return_sfc21 := FILL(BVAL := #fill_value_0, BLK    =>  "PAR_HTR_2_PWR");
       #return_sfc21 := FILL(BVAL := #fill_value_0, BLK    =>  "PAR_HTR_1_TMP");
       #return_sfc21 := FILL(BVAL := #fill_value_0, BLK    =>  "PAR_HTR_2_TMP");
       #return_sfc21 := FILL(BVAL := #fill_value_0, BLK    =>  "PAR_MAG_AV_CUR");
       #return_sfc21 := FILL(BVAL := #fill_value_1, BLK    =>  "PAR_MAG_RATIO_CUR");
       #return_sfc21 := FILL(BVAL := #fill_value_2, BLK    =>  "PAR_PRS");
       #return_sfc21 := FILL(BVAL := #fill_value_0, BLK    =>  "PAR_GAS_1_FLW");
       #return_sfc21 := FILL(BVAL := #fill_value_0, BLK    =>  "PAR_GAS_2_FLW");
       #return_sfc21 := FILL(BVAL := #fill_value_0, BLK    =>  "PAR_GAS_SUM_FLW");
       #return_sfc21 := FILL(BVAL := #fill_value_0, BLK    =>  "PAR_XT_DIA");
       #return_sfc21 := FILL(BVAL := #fill_value_0, BLK    =>  "PAR_AV_SPD");
       #return_sfc21 := FILL(BVAL := #fill_value_0, BLK    =>  "PAR_AV_SPD_DEV_1");
       #return_sfc21 := FILL(BVAL := #fill_value_0, BLK    =>  "PAR_AV_SPD_DEV_2");
       #return_sfc21 := FILL(BVAL := #fill_value_0, BLK    =>  "PAR_XT_GRO");
       #return_sfc21 := FILL(BVAL := #fill_value_0, BLK    =>  "PAR_MLT_TMP_1");
       #return_sfc21 := FILL(BVAL := #fill_value_0, BLK    =>  "PAR_MLT_LVL_INC");
       #return_sfc21 := FILL(BVAL := #fill_value_0, BLK    =>  "PAR_CTRL_DIA_GN");
       #return_sfc21 := FILL(BVAL := #fill_value_0, BLK    =>  "PAR_CTRL_DIA_TI");
       #return_sfc21 := FILL(BVAL := #fill_value_0, BLK    =>  "PAR_CTRL_DIA_TD");
       #return_sfc21 := FILL(BVAL := #fill_value_0, BLK    =>  "PAR_CTRL_DIA_T1");
       #return_sfc21 := FILL(BVAL := #fill_value_0, BLK    =>  "PAR_CTRL_DIA_TF");
       #return_sfc21 := FILL(BVAL := #fill_value_0, BLK    =>  "PAR_CTRL_GRO_GN");
       #return_sfc21 := FILL(BVAL := #fill_value_0, BLK    =>  "PAR_CTRL_GRO_TI");
       #return_sfc21 := FILL(BVAL := #fill_value_0, BLK    =>  "PAR_CTRL_GRO_TD");
       #return_sfc21 := FILL(BVAL := #fill_value_0, BLK    =>  "PAR_CTRL_GRO_T1");
       #return_sfc21 := FILL(BVAL := #fill_value_0, BLK    =>  "PAR_CTRL_GRO_TF");
       #return_sfc21 := FILL(BVAL := #fill_value_0, BLK    =>  "PAR_CTRL_AV_SPD_GN");
       #return_sfc21 := FILL(BVAL := #fill_value_0, BLK    =>  "PAR_CTRL_AV_SPD_TI");
       #return_sfc21 := FILL(BVAL := #fill_value_0, BLK    =>  "PAR_CTRL_AV_SPD_TD");
       #return_sfc21 := FILL(BVAL := #fill_value_0, BLK    =>  "PAR_CTRL_AV_SPD_T1");
       #return_sfc21 := FILL(BVAL := #fill_value_0, BLK    =>  "PAR_CTRL_AV_SPD_TF");
       #return_sfc21 := FILL(BVAL := #fill_value_0, BLK    =>  "PAR_CTRL_MLT_LVL_GN");
       #return_sfc21 := FILL(BVAL := #fill_value_0, BLK    =>  "PAR_CTRL_MLT_LVL_TI");
       #return_sfc21 := FILL(BVAL := #fill_value_0, BLK    =>  "PAR_CTRL_MLT_LVL_TD");
       #return_sfc21 := FILL(BVAL := #fill_value_0, BLK    =>  "PAR_CTRL_MLT_LVL_T1");
       #return_sfc21 := FILL(BVAL := #fill_value_0, BLK    =>  "PAR_CTRL_MLT_LVL_TF");
       #return_sfc21 := FILL(BVAL := #fill_value_0, BLK    =>  "PAR_CTRL_MLT_TMP_1_GN");
       #return_sfc21 := FILL(BVAL := #fill_value_0, BLK    =>  "PAR_CTRL_MLT_TMP_1_TI");
       #return_sfc21 := FILL(BVAL := #fill_value_0, BLK    =>  "PAR_CTRL_MLT_TMP_1_TD");
       #return_sfc21 := FILL(BVAL := #fill_value_0, BLK    =>  "PAR_CTRL_MLT_TMP_1_T1");
       #return_sfc21 := FILL(BVAL := #fill_value_0, BLK    =>  "PAR_CTRL_MLT_TMP_1_TF");
       #return_sfc21 := FILL(BVAL := #fill_value_0, BLK    =>  "PAR_CTRL_PRS_GN");
       #return_sfc21 := FILL(BVAL := #fill_value_0, BLK    =>  "PAR_CTRL_PRS_TI");
       #return_sfc21 := FILL(BVAL := #fill_value_0, BLK    =>  "PAR_CTRL_PRS_TD");
       #return_sfc21 := FILL(BVAL := #fill_value_0, BLK    =>  "PAR_CTRL_PRS_T1");
       #return_sfc21 := FILL(BVAL := #fill_value_0, BLK    =>  "PAR_CTRL_PRS_TF");
       #return_sfc21 := FILL(BVAL := #fill_value_0, BLK    =>  "PAR_XT_MEN");
       #return_sfc21 := FILL(BVAL := #fill_value_0, BLK    =>  "PAR_CR_CHARGE_WGT");
       #return_sfc21 := FILL(BVAL := #fill_value_0, BLK    =>  "PAR_CR_DIA");
       #return_sfc21 := FILL(BVAL := #fill_value_0, BLK    =>  "PAR_CR_FILL_LEVEL");
       #return_sfc21 := FILL(BVAL := #fill_value_0, BLK    =>  "PAR_TMP_COEFF_1");
       #return_sfc21 := FILL(BVAL := #fill_value_0, BLK    =>  "PAR_TMP_COEFF_2");
       #return_sfc21 := FILL(BVAL := #fill_value_0, BLK    =>  "PAR_PWR_COEFF_1");
       #return_sfc21 := FILL(BVAL := #fill_value_0, BLK    =>  "PAR_PWR_COEFF_2");
       #return_sfc21 := FILL(BVAL := #fill_value_0, BLK    =>  "PAR_CAM_THR");
       #return_sfc21 := FILL(BVAL := #fill_value_0, BLK    =>  "PAR_CAM_WIN_SIZE_H");
       #return_sfc21 := FILL(BVAL := #fill_value_0, BLK    =>  "PAR_CAM_WIN_SIZE_V");
       #return_sfc21 := FILL(BVAL := #fill_value_0, BLK    =>  "PAR_CAM_WIN_POS_H");
       #return_sfc21 := FILL(BVAL := #fill_value_0, BLK    =>  "PAR_CAM_WIN_POS_V");
       #return_sfc21 := FILL(BVAL := #fill_value_0, BLK    =>  "PAR_TME");
       #return_sfc21 := FILL(BVAL := #fill_value_0, BLK    =>  "PAR_X_VALUES_1");
       #return_sfc21 := FILL(BVAL := #fill_value_0, BLK    =>  "PAR_X_VALUES_2");
       #return_sfc21 := FILL(BVAL := #fill_value_0, BLK    =>  "PAR_X_VALUES_3");
       #return_sfc21 := FILL(BVAL := #fill_value_0, BLK    =>  "PAR_X_VALUES_4");
       #return_sfc21 := FILL(BVAL := #fill_value_0, BLK    =>  "PAR_X_VALUES_5");
       #return_sfc21 := FILL(BVAL := #fill_value_0, BLK    =>  "PAR_X_VALUES_6");
       #return_sfc21 := FILL(BVAL := #fill_value_0, BLK    =>  "PAR_X_VALUES_7");
       #return_sfc21 := FILL(BVAL := #fill_value_0, BLK    =>  "PAR_X_VALUES_8");
       #return_sfc21 := FILL(BVAL := #fill_value_0, BLK    =>  "PAR_X_VALUES_9");
       #return_sfc21 := FILL(BVAL := #fill_value_0, BLK    =>  "PAR_X_VALUES_10");
       #return_sfc21 := FILL(BVAL := #fill_value_0, BLK    =>  "PAR_AV_CRUC_ROT");
       #return_sfc21 := FILL(BVAL := #fill_value_0, BLK    =>  "PAR_AV_CRUC_ROT_DEV_1");
       #return_sfc21 := FILL(BVAL := #fill_value_0, BLK    =>  "PAR_AV_CRUC_ROT_DEV_2");    
       #return_sfc21 := FILL(BVAL := #fill_value_0, BLK    =>  "PAR_CTRL_AV_CRUC_ROT_GN");
       #return_sfc21 := FILL(BVAL := #fill_value_0, BLK    =>  "PAR_CTRL_AV_CRUC_ROT_TI");
       #return_sfc21 := FILL(BVAL := #fill_value_0, BLK    =>  "PAR_CTRL_AV_CRUC_ROT_TD");
       #return_sfc21 := FILL(BVAL := #fill_value_0, BLK    =>  "PAR_CTRL_AV_CRUC_ROT_T1"); 
       #return_sfc21 := FILL(BVAL := #fill_value_0, BLK    =>  "PAR_CR_ROT_RP_TME_UP");
       #return_sfc21 := FILL(BVAL := #fill_value_0, BLK    =>  "PAR_CR_ROT_RP_TME_DN");
       #return_sfc21 := FILL(BVAL := #fill_value_0, BLK    =>  "PAR_CAM_SET_OUT_RAD");
       #return_sfc21 := FILL(BVAL := #fill_value_0, BLK    =>  "PAR_CAM_SET_IN_RAD");
       #return_sfc21 := FILL(BVAL := #fill_value_0, BLK    =>  "PAR_CAM_SET_SEQ_STR_AGL");
       #return_sfc21 := FILL(BVAL := #fill_value_0, BLK    =>  "PAR_CAM_SET_SEQ_STP_AGL");

       #return_sfc21 := FILL(BVAL := #fill_value_0, BLK    =>  "APC");
       //return_sfc21 := FILL_SFC21(bval := fill_value_0, blk    :=  PDI);
       #return_sfc21 := FILL(BVAL := #fill_value_0, BLK    =>  "PDO");
       //return_sfc21 := FILL_SFC21(bval := fill_value_0, blk    :=  SDI);
       //return_sfc21 := FILL_SFC21(bval := fill_value_0, blk    :=  SDO);
       //return_sfc21 := FILL_SFC21(bval := fill_value_0, blk    :=  PAI);
       #return_sfc21 := FILL(BVAL := #fill_value_0, BLK    =>  "PAO");
       //return_sfc21 := FILL_SFC21(bval := fill_value_0, blk    :=  SAI);
       //return_sfc21 := FILL_SFC21(bval := fill_value_0, blk    :=  SAO);
       #return_sfc21 := FILL(BVAL := #fill_value_0, BLK    =>  "DV" );
       #return_sfc21 := FILL(BVAL := #fill_value_0, BLK    =>  "AV");
       #return_sfc21 := FILL(BVAL := #fill_value_0, BLK    =>  "DC");
       #return_sfc21 := FILL(BVAL := #fill_value_0, BLK    =>  "AC");
       //return_sfc21 := FILL_SFC21(bval := fill_value_0, blk    :=  FLT);
       #return_sfc21 := FILL(BVAL := #fill_value_0, BLK    =>  "SM_FLT_ACKN");
       #return_sfc21 := FILL(BVAL := #fill_value_0, BLK    =>  "KYD");
       //return_sfc21 := FILL_SFC21(bval := fill_value_0, blk    :=  LT);
       //return_sfc21 := FILL_SFC21(bval := fill_value_0, blk    :=  DIS);
       #return_sfc21 := FILL(BVAL := #fill_value_0, BLK    =>  "KYA");
       //return_sfc21 := FILL_SFC21(bval := fill_value_0, blk    :=  STA);
       #return_sfc21 := FILL(BVAL := #fill_value_0, BLK    =>  "SM_FLT_NOT_ACKN");
       //return_sfc21 := FILL_SFC21(bval := fill_value_0, blk    :=  AM_TEST_DB);
       #return_sfc21 := FILL(BVAL := #fill_value_0, BLK    =>  "BM_VAC_DB");
       #return_sfc21 := FILL(BVAL := #fill_value_0, BLK    =>  "CM_LOOP_PRS_DB");
       #return_sfc21 := FILL(BVAL := #fill_value_0, BLK    =>  "CM_LOOP_DIA_DB");
       #return_sfc21 := FILL(BVAL := #fill_value_0, BLK    =>  "CM_LOOP_HTR_1_DB");
       #return_sfc21 := FILL(BVAL := #fill_value_0, BLK    =>  "CM_LOOP_HTR_2_DB");
       #return_sfc21 := FILL(BVAL := #fill_value_0, BLK    =>  "CM_LOOP_AVG_SPD_DB");
       #return_sfc21 := FILL(BVAL := #fill_value_0, BLK    =>  "CM_LOOP_AVG_CRUC_ROT_DB");   
       #return_sfc21 := FILL(BVAL := #fill_value_0, BLK    =>  "CM_LOOP_MLT_TMP_DB");
       #return_sfc21 := FILL(BVAL := #fill_value_0, BLK    =>  "CM_LOOP_GRW_RTE_DB");
       #return_sfc21 := FILL(BVAL := #fill_value_0, BLK    =>  "CM_LOOP_MLT_LVL_DB");
       #return_sfc21 := FILL(BVAL := #fill_value_0, BLK    =>  "CM_AVG_MSR_SEN_POS_DB");
       #return_sfc21 := FILL(BVAL := #fill_value_0, BLK    =>  "CM_LOOP_MLT_DRIFT_DB");
       #return_sfc21 := FILL(BVAL := #fill_value_0, BLK    =>  "CM_LOOP_GAP_DB");
       #return_sfc21 := FILL(BVAL := #fill_value_0, BLK    =>  "CM_LOOP_AVG_GAP_OFFS_DB");

